LIN {X 0,Y 509.826,Z 394.48,A -85,B 0,C 180,E1 -5633.741,E2 -5633.741} C_VEL
LIN {X 0,Y 509.161,Z 394.559,A -85,B 0,C 180,E1 -5634.401,E2 -5634.401} C_VEL
LIN {X 0,Y 506.342,Z 394.916,A -85,B 0,C 180,E1 -5635.473,E2 -5635.473} C_VEL
LIN {X 0,Y 503.949,Z 395.212,A -85,B 0,C 180,E1 -5636.336,E2 -5636.336} C_VEL
LIN {X 0,Y 502.9,Z 395.339,A -85,B 0,C 180,E1 -5637.003,E2 -5637.003} C_VEL
LIN {X 0,Y 502.803,Z 395.349,A -85,B 0,C 180,E1 -5637.228,E2 -5637.228} C_VEL
LIN {X 0,Y 502.809,Z 395.349,A -85,B 0,C 180,E1 -5640.065,E2 -5640.065} C_VEL
LIN {X 0,Y 502.83,Z 395.345,A -85,B 0,C 180,E1 -5642.534,E2 -5642.534} C_VEL
LIN {X 0,Y 502.824,Z 395.354,A -85,B 0,C 180,E1 -5645.299,E2 -5645.299} C_VEL
LIN {X 0,Y 502.789,Z 395.353,A -85,B 0,C 180,E1 -5647.827,E2 -5647.827} C_VEL
LIN {X 0,Y 502.82,Z 395.346,A -85,B 0,C 180,E1 -5650.4,E2 -5650.4} C_VEL
LIN {X 0,Y 502.83,Z 395.351,A -85,B 0,C 180,E1 -5652.932,E2 -5652.932} C_VEL
LIN {X 0,Y 502.841,Z 395.351,A -85,B 0,C 180,E1 -5655.429,E2 -5655.429} C_VEL
LIN {X 0,Y 502.874,Z 395.344,A -85,B 0,C 180,E1 -5658.717,E2 -5658.717} C_VEL
LIN {X 0,Y 502.898,Z 395.34,A -85,B 0,C 180,E1 -5661.967,E2 -5661.967} C_VEL
LIN {X 0,Y 502.939,Z 395.335,A -85,B 0,C 180,E1 -5664.387,E2 -5664.387} C_VEL
LIN {X 0,Y 503.023,Z 395.325,A -85,B 0,C 180,E1 -5667.598,E2 -5667.598} C_VEL
LIN {X 0,Y 503.025,Z 395.324,A -85,B 0,C 180,E1 -5670,E2 -5670} C_VEL
LIN {X 0,Y 503.023,Z 395.325,A -85,B 0,C 180,E1 -5672.402,E2 -5672.402} C_VEL
LIN {X 0,Y 502.939,Z 395.335,A -85,B 0,C 180,E1 -5675.614,E2 -5675.614} C_VEL
LIN {X 0,Y 502.899,Z 395.339,A -85,B 0,C 180,E1 -5678.033,E2 -5678.033} C_VEL
LIN {X 0,Y 502.875,Z 395.344,A -85,B 0,C 180,E1 -5681.283,E2 -5681.283} C_VEL
LIN {X 0,Y 502.841,Z 395.351,A -85,B 0,C 180,E1 -5684.571,E2 -5684.571} C_VEL
LIN {X 0,Y 502.858,Z 395.344,A -85,B 0,C 180,E1 -5687.907,E2 -5687.907} C_VEL
LIN {X 0,Y 502.825,Z 395.353,A -85,B 0,C 180,E1 -5690.536,E2 -5690.536} C_VEL
LIN {X 0,Y 502.793,Z 395.353,A -85,B 0,C 180,E1 -5693.04,E2 -5693.04} C_VEL
LIN {X 0,Y 502.838,Z 395.344,A -85,B 0,C 180,E1 -5695.675,E2 -5695.675} C_VEL
LIN {X 0,Y 502.837,Z 395.35,A -85,B 0,C 180,E1 -5698.373,E2 -5698.373} C_VEL
LIN {X 0,Y 502.792,Z 395.35,A -85,B 0,C 180,E1 -5701.5,E2 -5701.5} C_VEL
LIN {X 0,Y 502.802,Z 395.358,A -85,B 0,C 180,E1 -5704.445,E2 -5704.445} C_VEL
LIN {X 0,Y 502.777,Z 395.352,A -85,B 0,C 180,E1 -5707.179,E2 -5707.179} C_VEL
LIN {X 0,Y 502.817,Z 395.35,A -85,B 0,C 180,E1 -5710.012,E2 -5710.012} C_VEL
LIN {X 0,Y 502.819,Z 395.353,A -85,B 0,C 180,E1 -5712.202,E2 -5712.202} C_VEL
LIN {X 0,Y 502.795,Z 395.35,A -85,B 0,C 180,E1 -5715.468,E2 -5715.468} C_VEL
LIN {X 0,Y 502.815,Z 395.348,A -85,B 0,C 180,E1 -5718.934,E2 -5718.934} C_VEL
LIN {X 0,Y 502.789,Z 395.357,A -85,B 0,C 180,E1 -5722.046,E2 -5722.046} C_VEL
LIN {X 0,Y 502.804,Z 395.349,A -85,B 0,C 180,E1 -5725.035,E2 -5725.035} C_VEL
LIN {X 0,Y 502.783,Z 395.357,A -85,B 0,C 180,E1 -5727.916,E2 -5727.916} C_VEL
LIN {X 0,Y 502.834,Z 395.346,A -85,B 0,C 180,E1 -5730.713,E2 -5730.713} C_VEL
LIN {X 0,Y 502.857,Z 395.343,A -85,B 0,C 180,E1 -5733.439,E2 -5733.439} C_VEL
LIN {X 0,Y 502.787,Z 395.358,A -85,B 0,C 180,E1 -5736.087,E2 -5736.087} C_VEL
LIN {X 0,Y 502.778,Z 395.352,A -85,B 0,C 180,E1 -5738.689,E2 -5738.689} C_VEL
LIN {X 0,Y 502.826,Z 395.347,A -85,B 0,C 180,E1 -5741.249,E2 -5741.249} C_VEL
LIN {X 0,Y 502.819,Z 395.354,A -85,B 0,C 180,E1 -5743.768,E2 -5743.768} C_VEL
LIN {X 0,Y 502.827,Z 395.349,A -85,B 0,C 180,E1 -5746.255,E2 -5746.255} C_VEL
LIN {X 0,Y 502.872,Z 395.34,A -85,B 0,C 180,E1 -5748.717,E2 -5748.717} C_VEL
LIN {X 0,Y 502.897,Z 395.342,A -85,B 0,C 180,E1 -5751.967,E2 -5751.967} C_VEL
LIN {X 0,Y 502.934,Z 395.333,A -85,B 0,C 180,E1 -5754.387,E2 -5754.387} C_VEL
LIN {X 0,Y 503.021,Z 395.33,A -85,B 0,C 180,E1 -5757.598,E2 -5757.598} C_VEL
LIN {X 0,Y 503.023,Z 395.325,A -85,B 0,C 180,E1 -5760,E2 -5760} C_VEL
LIN {X 0,Y 503.021,Z 395.322,A -85,B 0,C 180,E1 -5762.403,E2 -5762.403} C_VEL
LIN {X 0,Y 502.935,Z 395.34,A -85,B 0,C 180,E1 -5765.614,E2 -5765.614} C_VEL
LIN {X 0,Y 502.898,Z 395.339,A -85,B 0,C 180,E1 -5768.034,E2 -5768.034} C_VEL
LIN {X 0,Y 502.874,Z 395.346,A -85,B 0,C 180,E1 -5771.284,E2 -5771.284} C_VEL
LIN {X 0,Y 502.842,Z 395.344,A -85,B 0,C 180,E1 -5774.571,E2 -5774.571} C_VEL
LIN {X 0,Y 502.859,Z 395.343,A -85,B 0,C 180,E1 -5777.907,E2 -5777.907} C_VEL
LIN {X 0,Y 502.826,Z 395.346,A -85,B 0,C 180,E1 -5780.537,E2 -5780.537} C_VEL
LIN {X 0,Y 502.792,Z 395.356,A -85,B 0,C 180,E1 -5783.041,E2 -5783.041} C_VEL
LIN {X 0,Y 502.838,Z 395.347,A -85,B 0,C 180,E1 -5785.676,E2 -5785.676} C_VEL
LIN {X 0,Y 502.839,Z 395.345,A -85,B 0,C 180,E1 -5788.373,E2 -5788.373} C_VEL
LIN {X 0,Y 502.795,Z 395.353,A -85,B 0,C 180,E1 -5791.5,E2 -5791.5} C_VEL
LIN {X 0,Y 502.805,Z 395.35,A -85,B 0,C 180,E1 -5794.445,E2 -5794.445} C_VEL
LIN {X 0,Y 502.781,Z 395.36,A -85,B 0,C 180,E1 -5797.179,E2 -5797.179} C_VEL
LIN {X 0,Y 502.788,Z 395.355,A -85,B 0,C 180,E1 -5800.016,E2 -5800.016} C_VEL
LIN {X 0,Y 502.802,Z 395.354,A -85,B 0,C 180,E1 -5802.2,E2 -5802.2} C_VEL
LIN {X 0,Y 502.772,Z 395.36,A -85,B 0,C 180,E1 -5803.375,E2 -5803.375} C_VEL
LIN {X 0,Y 502.912,Z 396.072,A -85,B 0,C 180,E1 -5804.545,E2 -5804.545} C_VEL
LIN {X 0,Y 503.525,Z 400.319,A -85,B 0,C 180,E1 -5807.711,E2 -5807.711} C_VEL
LIN {X 0,Y 503.571,Z 403.923,A -85,B 0,C 180,E1 -5810.139,E2 -5810.139} C_VEL
LIN {X 0,Y 503.281,Z 408.665,A -85,B 0,C 180,E1 -5813.097,E2 -5813.097} C_VEL
LIN {X 0,Y 503.066,Z 413.701,A -85,B 0,C 180,E1 -5816.027,E2 -5816.027} C_VEL
LIN {X 0,Y 502.877,Z 418.836,A -85,B 0,C 180,E1 -5818.863,E2 -5818.863} C_VEL
LIN {X 0,Y 502.696,Z 424.321,A -85,B 0,C 180,E1 -5821.737,E2 -5821.737} C_VEL
LIN {X 0,Y 502.579,Z 429.398,A -85,B 0,C 180,E1 -5824.31,E2 -5824.31} C_VEL
LIN {X 0,Y 502.486,Z 435.794,A -85,B 0,C 180,E1 -5827.385,E2 -5827.385} C_VEL
LIN {X 0,Y 502.376,Z 442.071,A -85,B 0,C 180,E1 -5830.382,E2 -5830.382} C_VEL
LIN {X 0,Y 502.245,Z 447.46,A -85,B 0,C 180,E1 -5832.911,E2 -5832.911} C_VEL
LIN {X 0,Y 502.241,Z 453.523,A -85,B 0,C 180,E1 -5835.722,E2 -5835.722} C_VEL
LIN {X 0,Y 504.317,Z 465.721,A -85,B 0,C 180,E1 -5836.09,E2 -5836.09} C_VEL
LIN {X 0,Y 504.61,Z 469.05,A -85,B 0,C 180,E1 -5836.201,E2 -5836.201} C_VEL
LIN {X 0,Y 504.336,Z 481.375,A -85,B 0,C 180,E1 -5836.707,E2 -5836.707} C_VEL
LIN {X 0,Y 504.044,Z 491.745,A -85,B 0,C 180,E1 -5837.267,E2 -5837.267} C_VEL
LIN {X 0,Y 503.765,Z 501.474,A -85,B 0,C 180,E1 -5837.921,E2 -5837.921} C_VEL
LIN {X 0,Y 503.465,Z 510.173,A -85,B 0,C 180,E1 -5838.628,E2 -5838.628} C_VEL
LIN {X 0,Y 503.19,Z 517.54,A -85,B 0,C 180,E1 -5839.335,E2 -5839.335} C_VEL
LIN {X 0,Y 502.948,Z 524.728,A -85,B 0,C 180,E1 -5840.144,E2 -5840.144} C_VEL
LIN {X 0,Y 502.683,Z 532.274,A -85,B 0,C 180,E1 -5841.153,E2 -5841.153} C_VEL
LIN {X 0,Y 502.471,Z 538.564,A -85,B 0,C 180,E1 -5842.162,E2 -5842.162} C_VEL
LIN {X 0,Y 502.317,Z 543.988,A -85,B 0,C 180,E1 -5843.21,E2 -5843.21} C_VEL
LIN {X 0,Y 502.256,Z 548.894,A -85,B 0,C 180,E1 -5844.379,E2 -5844.379} C_VEL
LIN {X 0,Y 502.128,Z 552.85,A -85,B 0,C 180,E1 -5845.585,E2 -5845.585} C_VEL
LIN {X 0,Y 502.121,Z 555.772,A -85,B 0,C 180,E1 -5846.79,E2 -5846.79} C_VEL
LIN {X 0,Y 502.036,Z 558.196,A -85,B 0,C 180,E1 -5848.395,E2 -5848.395} C_VEL
LIN {X 0,Y 501.991,Z 558.78,A -85,B 0,C 180,E1 -5849.198,E2 -5849.198} C_VEL
LIN {X 0,Y 501.991,Z 558.78,A -85,B 0,C 180,E1 -5850.802,E2 -5850.802} C_VEL
LIN {X 0,Y 502.036,Z 558.196,A -85,B 0,C 180,E1 -5851.604,E2 -5851.604} C_VEL
LIN {X 0,Y 502.121,Z 555.772,A -85,B 0,C 180,E1 -5853.209,E2 -5853.209} C_VEL
LIN {X 0,Y 502.128,Z 552.851,A -85,B 0,C 180,E1 -5854.415,E2 -5854.415} C_VEL
LIN {X 0,Y 502.256,Z 548.896,A -85,B 0,C 180,E1 -5855.621,E2 -5855.621} C_VEL
LIN {X 0,Y 502.317,Z 543.989,A -85,B 0,C 180,E1 -5856.789,E2 -5856.789} C_VEL
LIN {X 0,Y 502.47,Z 538.566,A -85,B 0,C 180,E1 -5857.838,E2 -5857.838} C_VEL
LIN {X 0,Y 502.682,Z 532.277,A -85,B 0,C 180,E1 -5858.846,E2 -5858.846} C_VEL
LIN {X 0,Y 502.947,Z 524.731,A -85,B 0,C 180,E1 -5859.856,E2 -5859.856} C_VEL
LIN {X 0,Y 503.219,Z 515.622,A -85,B 0,C 180,E1 -5860.867,E2 -5860.867} C_VEL
LIN {X 0,Y 503.674,Z 504.176,A -85,B 0,C 180,E1 -5861.877,E2 -5861.877} C_VEL
LIN {X 0,Y 503.936,Z 494.382,A -85,B 0,C 180,E1 -5862.57,E2 -5862.57} C_VEL
LIN {X 0,Y 504.202,Z 484.399,A -85,B 0,C 180,E1 -5863.142,E2 -5863.142} C_VEL
LIN {X 0,Y 504.491,Z 474.335,A -85,B 0,C 180,E1 -5863.596,E2 -5863.596} C_VEL
LIN {X 0,Y 504.472,Z 466.607,A -85,B 0,C 180,E1 -5863.879,E2 -5863.879} C_VEL
LIN {X 0,Y 502.563,Z 455.442,A -85,B 0,C 180,E1 -5864.226,E2 -5864.226} C_VEL
LIN {X 0,Y 502.244,Z 453.524,A -85,B 0,C 180,E1 -5864.278,E2 -5864.278} C_VEL
LIN {X 0,Y 502.244,Z 447.461,A -85,B 0,C 180,E1 -5867.089,E2 -5867.089} C_VEL
LIN {X 0,Y 502.43,Z 440.391,A -85,B 0,C 180,E1 -5870.413,E2 -5870.413} C_VEL
LIN {X 0,Y 502.482,Z 434.885,A -85,B 0,C 180,E1 -5873.055,E2 -5873.055} C_VEL
LIN {X 0,Y 502.578,Z 429.398,A -85,B 0,C 180,E1 -5875.689,E2 -5875.689} C_VEL
LIN {X 0,Y 502.701,Z 424.094,A -85,B 0,C 180,E1 -5878.381,E2 -5878.381} C_VEL
LIN {X 0,Y 502.875,Z 418.832,A -85,B 0,C 180,E1 -5881.137,E2 -5881.137} C_VEL
LIN {X 0,Y 503.064,Z 413.669,A -85,B 0,C 180,E1 -5883.973,E2 -5883.973} C_VEL
LIN {X 0,Y 503.328,Z 408.065,A -85,B 0,C 180,E1 -5887.26,E2 -5887.26} C_VEL
LIN {X 0,Y 503.544,Z 403.787,A -85,B 0,C 180,E1 -5889.942,E2 -5889.942} C_VEL
LIN {X 0,Y 503.522,Z 400.313,A -85,B 0,C 180,E1 -5892.289,E2 -5892.289} C_VEL
LIN {X 0,Y 502.909,Z 396.09,A -85,B 0,C 180,E1 -5895.455,E2 -5895.455} C_VEL
LIN {X 0,Y 502.771,Z 395.359,A -85,B 0,C 180,E1 -5896.768,E2 -5896.768} C_VEL
LIN {X 0,Y 502.817,Z 395.356,A -85,B 0,C 180,E1 -5899.004,E2 -5899.004} C_VEL
LIN {X 0,Y 502.791,Z 395.353,A -85,B 0,C 180,E1 -5902.045,E2 -5902.045} C_VEL
LIN {X 0,Y 502.806,Z 395.357,A -85,B 0,C 180,E1 -5905.034,E2 -5905.034} C_VEL
LIN {X 0,Y 502.784,Z 395.351,A -85,B 0,C 180,E1 -5907.915,E2 -5907.915} C_VEL
LIN {X 0,Y 502.835,Z 395.352,A -85,B 0,C 180,E1 -5910.712,E2 -5910.712} C_VEL
LIN {X 0,Y 502.858,Z 395.343,A -85,B 0,C 180,E1 -5913.438,E2 -5913.438} C_VEL
LIN {X 0,Y 502.787,Z 395.352,A -85,B 0,C 180,E1 -5916.086,E2 -5916.086} C_VEL
LIN {X 0,Y 502.778,Z 395.36,A -85,B 0,C 180,E1 -5918.688,E2 -5918.688} C_VEL
LIN {X 0,Y 502.826,Z 395.347,A -85,B 0,C 180,E1 -5921.248,E2 -5921.248} C_VEL
LIN {X 0,Y 502.818,Z 395.347,A -85,B 0,C 180,E1 -5923.767,E2 -5923.767} C_VEL
LIN {X 0,Y 502.826,Z 395.35,A -85,B 0,C 180,E1 -5926.254,E2 -5926.254} C_VEL
LIN {X 0,Y 502.871,Z 395.347,A -85,B 0,C 180,E1 -5928.716,E2 -5928.716} C_VEL
LIN {X 0,Y 502.896,Z 395.339,A -85,B 0,C 180,E1 -5931.966,E2 -5931.966} C_VEL
LIN {X 0,Y 502.933,Z 395.34,A -85,B 0,C 180,E1 -5934.386,E2 -5934.386} C_VEL
LIN {X 0,Y 503.019,Z 395.322,A -85,B 0,C 180,E1 -5937.597,E2 -5937.597} C_VEL
LIN {X 0,Y 503.02,Z 395.325,A -85,B 0,C 180,E1 -5940,E2 -5940} C_VEL
LIN {X 0,Y 503.019,Z 395.33,A -85,B 0,C 180,E1 -5942.402,E2 -5942.402} C_VEL
LIN {X 0,Y 502.933,Z 395.333,A -85,B 0,C 180,E1 -5945.613,E2 -5945.613} C_VEL
LIN {X 0,Y 502.895,Z 395.343,A -85,B 0,C 180,E1 -5948.033,E2 -5948.033} C_VEL
LIN {X 0,Y 502.87,Z 395.34,A -85,B 0,C 180,E1 -5951.283,E2 -5951.283} C_VEL
LIN {X 0,Y 502.838,Z 395.347,A -85,B 0,C 180,E1 -5954.571,E2 -5954.571} C_VEL
LIN {X 0,Y 502.854,Z 395.348,A -85,B 0,C 180,E1 -5957.907,E2 -5957.907} C_VEL
LIN {X 0,Y 502.82,Z 395.349,A -85,B 0,C 180,E1 -5960.536,E2 -5960.536} C_VEL
LIN {X 0,Y 502.789,Z 395.35,A -85,B 0,C 180,E1 -5963.04,E2 -5963.04} C_VEL
LIN {X 0,Y 502.834,Z 395.349,A -85,B 0,C 180,E1 -5965.675,E2 -5965.675} C_VEL
LIN {X 0,Y 502.835,Z 395.348,A -85,B 0,C 180,E1 -5968.372,E2 -5968.372} C_VEL
LIN {X 0,Y 502.79,Z 395.354,A -85,B 0,C 180,E1 -5971.5,E2 -5971.5} C_VEL
LIN {X 0,Y 502.8,Z 395.351,A -85,B 0,C 180,E1 -5974.445,E2 -5974.445} C_VEL
LIN {X 0,Y 502.774,Z 395.353,A -85,B 0,C 180,E1 -5977.178,E2 -5977.178} C_VEL
LIN {X 0,Y 502.819,Z 395.352,A -85,B 0,C 180,E1 -5980.012,E2 -5980.012} C_VEL
LIN {X 0,Y 502.822,Z 395.349,A -85,B 0,C 180,E1 -5982.203,E2 -5982.203} C_VEL
LIN {X 0,Y 502.794,Z 395.355,A -85,B 0,C 180,E1 -5985.468,E2 -5985.468} C_VEL
LIN {X 0,Y 502.829,Z 395.351,A -85,B 0,C 180,E1 -5987.865,E2 -5987.865} C_VEL
LIN {X 0,Y 502.803,Z 395.35,A -85,B 0,C 180,E1 -5991.025,E2 -5991.025} C_VEL
LIN {X 0,Y 502.78,Z 395.353,A -85,B 0,C 180,E1 -5994.167,E2 -5994.167} C_VEL
LIN {X 0,Y 502.803,Z 395.349,A -85,B 0,C 180,E1 -5997.228,E2 -5997.228} C_VEL
LIN {X 0,Y 502.104,Z 395.439,A -85,B 0,C 180,E1 -5997.897,E2 -5997.897} C_VEL
LIN {X 0,Y 499.238,Z 395.795,A -85,B 0,C 180,E1 -5998.983,E2 -5998.983} C_VEL
LIN {X 0,Y 496.842,Z 396.095,A -85,B 0,C 180,E1 -5999.858,E2 -5999.858} C_VEL
LIN {X 0,Y 495.826,Z 396.218,A -85,B 0,C 180,E1 -6000.533,E2 -6000.533} C_VEL
LIN {X 0,Y 495.748,Z 396.228,A -85,B 0,C 180,E1 -6000.762,E2 -6000.762} C_VEL
LIN {X 0,Y 495.794,Z 396.224,A -85,B 0,C 180,E1 -6003.933,E2 -6003.933} C_VEL
LIN {X 0,Y 495.753,Z 396.232,A -85,B 0,C 180,E1 -6007.14,E2 -6007.14} C_VEL
LIN {X 0,Y 495.773,Z 396.225,A -85,B 0,C 180,E1 -6010.11,E2 -6010.11} C_VEL
LIN {X 0,Y 495.782,Z 396.227,A -85,B 0,C 180,E1 -6012.682,E2 -6012.682} C_VEL
LIN {X 0,Y 495.786,Z 396.232,A -85,B 0,C 180,E1 -6015.217,E2 -6015.217} C_VEL
LIN {X 0,Y 495.848,Z 396.218,A -85,B 0,C 180,E1 -6018.555,E2 -6018.555} C_VEL
LIN {X 0,Y 495.87,Z 396.216,A -85,B 0,C 180,E1 -6021.852,E2 -6021.852} C_VEL
LIN {X 0,Y 495.896,Z 396.212,A -85,B 0,C 180,E1 -6024.307,E2 -6024.307} C_VEL
LIN {X 0,Y 495.991,Z 396.202,A -85,B 0,C 180,E1 -6027.564,E2 -6027.564} C_VEL
LIN {X 0,Y 495.996,Z 396.2,A -85,B 0,C 180,E1 -6030,E2 -6030} C_VEL
LIN {X 0,Y 495.992,Z 396.202,A -85,B 0,C 180,E1 -6032.436,E2 -6032.436} C_VEL
LIN {X 0,Y 495.897,Z 396.212,A -85,B 0,C 180,E1 -6035.694,E2 -6035.694} C_VEL
LIN {X 0,Y 495.87,Z 396.216,A -85,B 0,C 180,E1 -6038.148,E2 -6038.148} C_VEL
LIN {X 0,Y 495.849,Z 396.218,A -85,B 0,C 180,E1 -6041.445,E2 -6041.445} C_VEL
LIN {X 0,Y 495.787,Z 396.232,A -85,B 0,C 180,E1 -6044.783,E2 -6044.783} C_VEL
LIN {X 0,Y 495.783,Z 396.227,A -85,B 0,C 180,E1 -6047.319,E2 -6047.319} C_VEL
LIN {X 0,Y 495.774,Z 396.225,A -85,B 0,C 180,E1 -6049.89,E2 -6049.89} C_VEL
LIN {X 0,Y 495.754,Z 396.232,A -85,B 0,C 180,E1 -6052.86,E2 -6052.86} C_VEL
LIN {X 0,Y 495.796,Z 396.224,A -85,B 0,C 180,E1 -6056.067,E2 -6056.067} C_VEL
LIN {X 0,Y 495.769,Z 396.23,A -85,B 0,C 180,E1 -6058.815,E2 -6058.815} C_VEL
LIN {X 0,Y 495.754,Z 396.227,A -85,B 0,C 180,E1 -6061.726,E2 -6061.726} C_VEL
LIN {X 0,Y 495.772,Z 396.23,A -85,B 0,C 180,E1 -6064.695,E2 -6064.695} C_VEL
LIN {X 0,Y 495.727,Z 396.23,A -85,B 0,C 180,E1 -6067.561,E2 -6067.561} C_VEL
LIN {X 0,Y 495.775,Z 396.228,A -85,B 0,C 180,E1 -6070.699,E2 -6070.699} C_VEL
LIN {X 0,Y 495.73,Z 396.231,A -85,B 0,C 180,E1 -6073.696,E2 -6073.696} C_VEL
LIN {X 0,Y 495.723,Z 396.239,A -85,B 0,C 180,E1 -6076.305,E2 -6076.305} C_VEL
LIN {X 0,Y 495.762,Z 396.226,A -85,B 0,C 180,E1 -6079.3,E2 -6079.3} C_VEL
LIN {X 0,Y 495.727,Z 396.235,A -85,B 0,C 180,E1 -6082.439,E2 -6082.439} C_VEL
LIN {X 0,Y 495.78,Z 396.224,A -85,B 0,C 180,E1 -6085.458,E2 -6085.458} C_VEL
LIN {X 0,Y 495.755,Z 396.232,A -85,B 0,C 180,E1 -6088.364,E2 -6088.364} C_VEL
LIN {X 0,Y 495.785,Z 396.225,A -85,B 0,C 180,E1 -6091.506,E2 -6091.506} C_VEL
LIN {X 0,Y 495.786,Z 396.23,A -85,B 0,C 180,E1 -6093.932,E2 -6093.932} C_VEL
LIN {X 0,Y 495.76,Z 396.226,A -85,B 0,C 180,E1 -6097.138,E2 -6097.138} C_VEL
LIN {X 0,Y 495.767,Z 396.231,A -85,B 0,C 180,E1 -6100.11,E2 -6100.11} C_VEL
LIN {X 0,Y 495.783,Z 396.223,A -85,B 0,C 180,E1 -6102.682,E2 -6102.682} C_VEL
LIN {X 0,Y 495.785,Z 396.224,A -85,B 0,C 180,E1 -6105.218,E2 -6105.218} C_VEL
LIN {X 0,Y 495.847,Z 396.216,A -85,B 0,C 180,E1 -6108.555,E2 -6108.555} C_VEL
LIN {X 0,Y 495.869,Z 396.22,A -85,B 0,C 180,E1 -6111.852,E2 -6111.852} C_VEL
LIN {X 0,Y 495.892,Z 396.211,A -85,B 0,C 180,E1 -6114.307,E2 -6114.307} C_VEL
LIN {X 0,Y 495.989,Z 396.205,A -85,B 0,C 180,E1 -6117.564,E2 -6117.564} C_VEL
LIN {X 0,Y 495.994,Z 396.2,A -85,B 0,C 180,E1 -6120,E2 -6120} C_VEL
LIN {X 0,Y 495.99,Z 396.198,A -85,B 0,C 180,E1 -6122.437,E2 -6122.437} C_VEL
LIN {X 0,Y 495.893,Z 396.216,A -85,B 0,C 180,E1 -6125.694,E2 -6125.694} C_VEL
LIN {X 0,Y 495.87,Z 396.213,A -85,B 0,C 180,E1 -6128.148,E2 -6128.148} C_VEL
LIN {X 0,Y 495.848,Z 396.224,A -85,B 0,C 180,E1 -6131.446,E2 -6131.446} C_VEL
LIN {X 0,Y 495.787,Z 396.224,A -85,B 0,C 180,E1 -6134.783,E2 -6134.783} C_VEL
LIN {X 0,Y 495.785,Z 396.232,A -85,B 0,C 180,E1 -6137.319,E2 -6137.319} C_VEL
LIN {X 0,Y 495.769,Z 396.226,A -85,B 0,C 180,E1 -6139.891,E2 -6139.891} C_VEL
LIN {X 0,Y 495.759,Z 396.229,A -85,B 0,C 180,E1 -6142.862,E2 -6142.862} C_VEL
LIN {X 0,Y 495.789,Z 396.223,A -85,B 0,C 180,E1 -6146.068,E2 -6146.068} C_VEL
LIN {X 0,Y 495.77,Z 396.229,A -85,B 0,C 180,E1 -6148.815,E2 -6148.815} C_VEL
LIN {X 0,Y 495.757,Z 396.228,A -85,B 0,C 180,E1 -6151.727,E2 -6151.727} C_VEL
LIN {X 0,Y 495.775,Z 396.228,A -85,B 0,C 180,E1 -6154.696,E2 -6154.696} C_VEL
LIN {X 0,Y 495.731,Z 396.235,A -85,B 0,C 180,E1 -6157.562,E2 -6157.562} C_VEL
LIN {X 0,Y 495.767,Z 396.233,A -85,B 0,C 180,E1 -6160.7,E2 -6160.7} C_VEL
LIN {X 0,Y 495.748,Z 396.299,A -85,B 0,C 180,E1 -6163.698,E2 -6163.698} C_VEL
LIN {X 0,Y 496.26,Z 399.542,A -85,B 0,C 180,E1 -6166.242,E2 -6166.242} C_VEL
LIN {X 0,Y 496.607,Z 402.78,A -85,B 0,C 180,E1 -6168.596,E2 -6168.596} C_VEL
LIN {X 0,Y 496.465,Z 407.14,A -85,B 0,C 180,E1 -6171.475,E2 -6171.475} C_VEL
LIN {X 0,Y 496.125,Z 412.071,A -85,B 0,C 180,E1 -6174.494,E2 -6174.494} C_VEL
LIN {X 0,Y 495.938,Z 417.147,A -85,B 0,C 180,E1 -6177.419,E2 -6177.419} C_VEL
LIN {X 0,Y 495.752,Z 422.337,A -85,B 0,C 180,E1 -6180.253,E2 -6180.253} C_VEL
LIN {X 0,Y 495.609,Z 428.151,A -85,B 0,C 180,E1 -6183.301,E2 -6183.301} C_VEL
LIN {X 0,Y 495.465,Z 432.972,A -85,B 0,C 180,E1 -6185.71,E2 -6185.71} C_VEL
LIN {X 0,Y 495.402,Z 438.478,A -85,B 0,C 180,E1 -6188.356,E2 -6188.356} C_VEL
LIN {X 0,Y 495.277,Z 443.867,A -85,B 0,C 180,E1 -6190.951,E2 -6190.951} C_VEL
LIN {X 0,Y 495.143,Z 449.257,A -85,B 0,C 180,E1 -6193.508,E2 -6193.508} C_VEL
LIN {X 0,Y 495.174,Z 453.523,A -85,B 0,C 180,E1 -6195.514,E2 -6195.514} C_VEL
LIN {X 0,Y 497.243,Z 465.704,A -85,B 0,C 180,E1 -6195.889,E2 -6195.889} C_VEL
LIN {X 0,Y 497.737,Z 469.054,A -85,B 0,C 180,E1 -6196.007,E2 -6196.007} C_VEL
LIN {X 0,Y 497.444,Z 481.366,A -85,B 0,C 180,E1 -6196.519,E2 -6196.519} C_VEL
LIN {X 0,Y 497.093,Z 491.986,A -85,B 0,C 180,E1 -6197.101,E2 -6197.101} C_VEL
LIN {X 0,Y 496.807,Z 501.467,A -85,B 0,C 180,E1 -6197.749,E2 -6197.749} C_VEL
LIN {X 0,Y 496.491,Z 510.167,A -85,B 0,C 180,E1 -6198.466,E2 -6198.466} C_VEL
LIN {X 0,Y 496.186,Z 517.535,A -85,B 0,C 180,E1 -6199.183,E2 -6199.183} C_VEL
LIN {X 0,Y 495.929,Z 524.724,A -85,B 0,C 180,E1 -6200.003,E2 -6200.003} C_VEL
LIN {X 0,Y 495.634,Z 532.27,A -85,B 0,C 180,E1 -6201.026,E2 -6201.026} C_VEL
LIN {X 0,Y 495.404,Z 538.559,A -85,B 0,C 180,E1 -6202.049,E2 -6202.049} C_VEL
LIN {X 0,Y 495.248,Z 543.983,A -85,B 0,C 180,E1 -6203.113,E2 -6203.113} C_VEL
LIN {X 0,Y 495.174,Z 548.89,A -85,B 0,C 180,E1 -6204.298,E2 -6204.298} C_VEL
LIN {X 0,Y 495.029,Z 552.846,A -85,B 0,C 180,E1 -6205.521,E2 -6205.521} C_VEL
LIN {X 0,Y 495.043,Z 555.769,A -85,B 0,C 180,E1 -6206.744,E2 -6206.744} C_VEL
LIN {X 0,Y 494.961,Z 558.195,A -85,B 0,C 180,E1 -6208.373,E2 -6208.373} C_VEL
LIN {X 0,Y 494.911,Z 558.779,A -85,B 0,C 180,E1 -6209.186,E2 -6209.186} C_VEL
LIN {X 0,Y 494.911,Z 558.78,A -85,B 0,C 180,E1 -6210.813,E2 -6210.813} C_VEL
LIN {X 0,Y 494.961,Z 558.195,A -85,B 0,C 180,E1 -6211.627,E2 -6211.627} C_VEL
LIN {X 0,Y 495.043,Z 555.77,A -85,B 0,C 180,E1 -6213.255,E2 -6213.255} C_VEL
LIN {X 0,Y 495.028,Z 552.847,A -85,B 0,C 180,E1 -6214.478,E2 -6214.478} C_VEL
LIN {X 0,Y 495.175,Z 548.891,A -85,B 0,C 180,E1 -6215.702,E2 -6215.702} C_VEL
LIN {X 0,Y 495.247,Z 543.985,A -85,B 0,C 180,E1 -6216.887,E2 -6216.887} C_VEL
LIN {X 0,Y 495.403,Z 538.561,A -85,B 0,C 180,E1 -6217.95,E2 -6217.95} C_VEL
LIN {X 0,Y 495.634,Z 532.272,A -85,B 0,C 180,E1 -6218.973,E2 -6218.973} C_VEL
LIN {X 0,Y 495.929,Z 524.727,A -85,B 0,C 180,E1 -6219.997,E2 -6219.997} C_VEL
LIN {X 0,Y 496.243,Z 515.62,A -85,B 0,C 180,E1 -6221.022,E2 -6221.022} C_VEL
LIN {X 0,Y 496.723,Z 504.168,A -85,B 0,C 180,E1 -6222.045,E2 -6222.045} C_VEL
LIN {X 0,Y 496.982,Z 494.866,A -85,B 0,C 180,E1 -6222.718,E2 -6222.718} C_VEL
LIN {X 0,Y 497.274,Z 484.389,A -85,B 0,C 180,E1 -6223.329,E2 -6223.329} C_VEL
LIN {X 0,Y 497.606,Z 474.326,A -85,B 0,C 180,E1 -6223.788,E2 -6223.788} C_VEL
LIN {X 0,Y 497.545,Z 467.464,A -85,B 0,C 180,E1 -6224.05,E2 -6224.05} C_VEL
LIN {X 0,Y 495.519,Z 455.49,A -85,B 0,C 180,E1 -6224.431,E2 -6224.431} C_VEL
LIN {X 0,Y 495.167,Z 453.524,A -85,B 0,C 180,E1 -6224.486,E2 -6224.486} C_VEL
LIN {X 0,Y 495.217,Z 445.99,A -85,B 0,C 180,E1 -6228.038,E2 -6228.038} C_VEL
LIN {X 0,Y 495.377,Z 440.275,A -85,B 0,C 180,E1 -6230.773,E2 -6230.773} C_VEL
LIN {X 0,Y 495.43,Z 434.813,A -85,B 0,C 180,E1 -6233.403,E2 -6233.403} C_VEL
LIN {X 0,Y 495.538,Z 429.353,A -85,B 0,C 180,E1 -6236.082,E2 -6236.082} C_VEL
LIN {X 0,Y 495.675,Z 424.091,A -85,B 0,C 180,E1 -6238.82,E2 -6238.82} C_VEL
LIN {X 0,Y 495.868,Z 418.623,A -85,B 0,C 180,E1 -6241.746,E2 -6241.746} C_VEL
LIN {X 0,Y 496.077,Z 413.358,A -85,B 0,C 180,E1 -6244.745,E2 -6244.745} C_VEL
LIN {X 0,Y 496.33,Z 408.7,A -85,B 0,C 180,E1 -6247.537,E2 -6247.537} C_VEL
LIN {X 0,Y 496.534,Z 404.625,A -85,B 0,C 180,E1 -6250.153,E2 -6250.153} C_VEL
LIN {X 0,Y 496.584,Z 402.356,A -85,B 0,C 180,E1 -6251.695,E2 -6251.695} C_VEL
LIN {X 0,Y 496.224,Z 399.276,A -85,B 0,C 180,E1 -6253.945,E2 -6253.945} C_VEL
LIN {X 0,Y 495.746,Z 396.296,A -85,B 0,C 180,E1 -6256.302,E2 -6256.302} C_VEL
LIN {X 0,Y 495.764,Z 396.233,A -85,B 0,C 180,E1 -6259.299,E2 -6259.299} C_VEL
LIN {X 0,Y 495.729,Z 396.235,A -85,B 0,C 180,E1 -6262.438,E2 -6262.438} C_VEL
LIN {X 0,Y 495.782,Z 396.226,A -85,B 0,C 180,E1 -6265.457,E2 -6265.457} C_VEL
LIN {X 0,Y 495.756,Z 396.229,A -85,B 0,C 180,E1 -6268.363,E2 -6268.363} C_VEL
LIN {X 0,Y 495.786,Z 396.224,A -85,B 0,C 180,E1 -6271.505,E2 -6271.505} C_VEL
LIN {X 0,Y 495.786,Z 396.223,A -85,B 0,C 180,E1 -6273.931,E2 -6273.931} C_VEL
LIN {X 0,Y 495.756,Z 396.23,A -85,B 0,C 180,E1 -6277.138,E2 -6277.138} C_VEL
LIN {X 0,Y 495.767,Z 396.227,A -85,B 0,C 180,E1 -6280.109,E2 -6280.109} C_VEL
LIN {X 0,Y 495.783,Z 396.232,A -85,B 0,C 180,E1 -6282.681,E2 -6282.681} C_VEL
LIN {X 0,Y 495.784,Z 396.224,A -85,B 0,C 180,E1 -6285.217,E2 -6285.217} C_VEL
LIN {X 0,Y 495.845,Z 396.224,A -85,B 0,C 180,E1 -6288.554,E2 -6288.554} C_VEL
LIN {X 0,Y 495.867,Z 396.214,A -85,B 0,C 180,E1 -6291.852,E2 -6291.852} C_VEL
LIN {X 0,Y 495.89,Z 396.216,A -85,B 0,C 180,E1 -6294.306,E2 -6294.306} C_VEL
LIN {X 0,Y 495.988,Z 396.198,A -85,B 0,C 180,E1 -6297.563,E2 -6297.563} C_VEL
LIN {X 0,Y 495.991,Z 396.201,A -85,B 0,C 180,E1 -6300,E2 -6300} C_VEL
LIN {X 0,Y 495.987,Z 396.205,A -85,B 0,C 180,E1 -6302.436,E2 -6302.436} C_VEL
LIN {X 0,Y 495.89,Z 396.211,A -85,B 0,C 180,E1 -6305.693,E2 -6305.693} C_VEL
LIN {X 0,Y 495.866,Z 396.22,A -85,B 0,C 180,E1 -6308.148,E2 -6308.148} C_VEL
LIN {X 0,Y 495.844,Z 396.216,A -85,B 0,C 180,E1 -6311.445,E2 -6311.445} C_VEL
LIN {X 0,Y 495.783,Z 396.224,A -85,B 0,C 180,E1 -6314.783,E2 -6314.783} C_VEL
LIN {X 0,Y 495.78,Z 396.224,A -85,B 0,C 180,E1 -6317.318,E2 -6317.318} C_VEL
LIN {X 0,Y 495.764,Z 396.231,A -85,B 0,C 180,E1 -6319.89,E2 -6319.89} C_VEL
LIN {X 0,Y 495.757,Z 396.227,A -85,B 0,C 180,E1 -6322.862,E2 -6322.862} C_VEL
LIN {X 0,Y 495.792,Z 396.23,A -85,B 0,C 180,E1 -6326.067,E2 -6326.067} C_VEL
LIN {X 0,Y 495.773,Z 396.225,A -85,B 0,C 180,E1 -6328.814,E2 -6328.814} C_VEL
LIN {X 0,Y 495.752,Z 396.233,A -85,B 0,C 180,E1 -6331.726,E2 -6331.726} C_VEL
LIN {X 0,Y 495.77,Z 396.225,A -85,B 0,C 180,E1 -6334.695,E2 -6334.695} C_VEL
LIN {X 0,Y 495.726,Z 396.235,A -85,B 0,C 180,E1 -6337.561,E2 -6337.561} C_VEL
LIN {X 0,Y 495.786,Z 396.227,A -85,B 0,C 180,E1 -6340.052,E2 -6340.052} C_VEL
LIN {X 0,Y 495.757,Z 396.227,A -85,B 0,C 180,E1 -6342.879,E2 -6342.879} C_VEL
LIN {X 0,Y 495.73,Z 396.234,A -85,B 0,C 180,E1 -6346,E2 -6346} C_VEL
LIN {X 0,Y 495.762,Z 396.226,A -85,B 0,C 180,E1 -6348.705,E2 -6348.705} C_VEL
LIN {X 0,Y 495.749,Z 396.233,A -85,B 0,C 180,E1 -6351.409,E2 -6351.409} C_VEL
LIN {X 0,Y 495.752,Z 396.227,A -85,B 0,C 180,E1 -6354.463,E2 -6354.463} C_VEL
LIN {X 0,Y 495.764,Z 396.233,A -85,B 0,C 180,E1 -6357.406,E2 -6357.406} C_VEL
LIN {X 0,Y 495.761,Z 396.226,A -85,B 0,C 180,E1 -6360.254,E2 -6360.254} C_VEL
LIN {X 0,Y 495.748,Z 396.228,A -85,B 0,C 180,E1 -6360.762,E2 -6360.762} C_VEL
LIN {X 0,Y 495.092,Z 396.318,A -85,B 0,C 180,E1 -6361.441,E2 -6361.441} C_VEL
LIN {X 0,Y 492.24,Z 396.669,A -85,B 0,C 180,E1 -6362.544,E2 -6362.544} C_VEL
LIN {X 0,Y 489.833,Z 396.973,A -85,B 0,C 180,E1 -6363.432,E2 -6363.432} C_VEL
LIN {X 0,Y 488.815,Z 397.092,A -85,B 0,C 180,E1 -6364.119,E2 -6364.119} C_VEL
LIN {X 0,Y 488.742,Z 397.1,A -85,B 0,C 180,E1 -6364.351,E2 -6364.351} C_VEL
LIN {X 0,Y 488.716,Z 397.109,A -85,B 0,C 180,E1 -6367.153,E2 -6367.153} C_VEL
LIN {X 0,Y 488.724,Z 397.106,A -85,B 0,C 180,E1 -6369.811,E2 -6369.811} C_VEL
LIN {X 0,Y 488.729,Z 397.104,A -85,B 0,C 180,E1 -6372.424,E2 -6372.424} C_VEL
LIN {X 0,Y 488.758,Z 397.106,A -85,B 0,C 180,E1 -6375,E2 -6375} C_VEL
LIN {X 0,Y 488.802,Z 397.095,A -85,B 0,C 180,E1 -6378.388,E2 -6378.388} C_VEL
LIN {X 0,Y 488.814,Z 397.096,A -85,B 0,C 180,E1 -6381.734,E2 -6381.734} C_VEL
LIN {X 0,Y 488.855,Z 397.089,A -85,B 0,C 180,E1 -6384.225,E2 -6384.225} C_VEL
LIN {X 0,Y 488.959,Z 397.078,A -85,B 0,C 180,E1 -6387.529,E2 -6387.529} C_VEL
LIN {X 0,Y 488.951,Z 397.081,A -85,B 0,C 180,E1 -6390.824,E2 -6390.824} C_VEL
LIN {X 0,Y 488.959,Z 397.078,A -85,B 0,C 180,E1 -6392.472,E2 -6392.472} C_VEL
LIN {X 0,Y 488.856,Z 397.089,A -85,B 0,C 180,E1 -6395.776,E2 -6395.776} C_VEL
LIN {X 0,Y 488.815,Z 397.095,A -85,B 0,C 180,E1 -6398.266,E2 -6398.266} C_VEL
LIN {X 0,Y 488.802,Z 397.095,A -85,B 0,C 180,E1 -6401.613,E2 -6401.613} C_VEL
LIN {X 0,Y 488.758,Z 397.106,A -85,B 0,C 180,E1 -6405,E2 -6405} C_VEL
LIN {X 0,Y 488.751,Z 397.105,A -85,B 0,C 180,E1 -6408.442,E2 -6408.442} C_VEL
LIN {X 0,Y 488.704,Z 397.108,A -85,B 0,C 180,E1 -6411.071,E2 -6411.071} C_VEL
LIN {X 0,Y 488.69,Z 397.107,A -85,B 0,C 180,E1 -6413.745,E2 -6413.745} C_VEL
LIN {X 0,Y 488.795,Z 397.097,A -85,B 0,C 180,E1 -6416.945,E2 -6416.945} C_VEL
LIN {X 0,Y 488.706,Z 397.111,A -85,B 0,C 180,E1 -6420.363,E2 -6420.363} C_VEL
LIN {X 0,Y 488.731,Z 397.102,A -85,B 0,C 180,E1 -6423.485,E2 -6423.485} C_VEL
LIN {X 0,Y 488.685,Z 397.115,A -85,B 0,C 180,E1 -6426.356,E2 -6426.356} C_VEL
LIN {X 0,Y 488.738,Z 397.101,A -85,B 0,C 180,E1 -6429.25,E2 -6429.25} C_VEL
LIN {X 0,Y 488.727,Z 397.108,A -85,B 0,C 180,E1 -6432.521,E2 -6432.521} C_VEL
LIN {X 0,Y 488.707,Z 397.105,A -85,B 0,C 180,E1 -6435.199,E2 -6435.199} C_VEL
LIN {X 0,Y 488.703,Z 397.112,A -85,B 0,C 180,E1 -6438.4,E2 -6438.4} C_VEL
LIN {X 0,Y 488.699,Z 397.106,A -85,B 0,C 180,E1 -6440.947,E2 -6440.947} C_VEL
LIN {X 0,Y 488.68,Z 397.112,A -85,B 0,C 180,E1 -6443.869,E2 -6443.869} C_VEL
LIN {X 0,Y 488.734,Z 397.102,A -85,B 0,C 180,E1 -6446.878,E2 -6446.878} C_VEL
LIN {X 0,Y 488.729,Z 397.106,A -85,B 0,C 180,E1 -6449.782,E2 -6449.782} C_VEL
LIN {X 0,Y 488.787,Z 397.095,A -85,B 0,C 180,E1 -6453.057,E2 -6453.057} C_VEL
LIN {X 0,Y 488.689,Z 397.112,A -85,B 0,C 180,E1 -6456.255,E2 -6456.255} C_VEL
LIN {X 0,Y 488.741,Z 397.101,A -85,B 0,C 180,E1 -6459.176,E2 -6459.176} C_VEL
LIN {X 0,Y 488.73,Z 397.104,A -85,B 0,C 180,E1 -6462.424,E2 -6462.424} C_VEL
LIN {X 0,Y 488.757,Z 397.099,A -85,B 0,C 180,E1 -6465,E2 -6465} C_VEL
LIN {X 0,Y 488.801,Z 397.094,A -85,B 0,C 180,E1 -6468.388,E2 -6468.388} C_VEL
LIN {X 0,Y 488.814,Z 397.1,A -85,B 0,C 180,E1 -6471.734,E2 -6471.734} C_VEL
LIN {X 0,Y 488.851,Z 397.089,A -85,B 0,C 180,E1 -6474.225,E2 -6474.225} C_VEL
LIN {X 0,Y 488.957,Z 397.08,A -85,B 0,C 180,E1 -6477.529,E2 -6477.529} C_VEL
LIN {X 0,Y 488.951,Z 397.075,A -85,B 0,C 180,E1 -6480.824,E2 -6480.824} C_VEL
LIN {X 0,Y 488.958,Z 397.073,A -85,B 0,C 180,E1 -6482.472,E2 -6482.472} C_VEL
LIN {X 0,Y 488.852,Z 397.092,A -85,B 0,C 180,E1 -6485.776,E2 -6485.776} C_VEL
LIN {X 0,Y 488.814,Z 397.092,A -85,B 0,C 180,E1 -6488.267,E2 -6488.267} C_VEL
LIN {X 0,Y 488.802,Z 397.099,A -85,B 0,C 180,E1 -6491.613,E2 -6491.613} C_VEL
LIN {X 0,Y 488.759,Z 397.102,A -85,B 0,C 180,E1 -6495.001,E2 -6495.001} C_VEL
LIN {X 0,Y 488.752,Z 397.099,A -85,B 0,C 180,E1 -6498.443,E2 -6498.443} C_VEL
LIN {X 0,Y 488.704,Z 397.11,A -85,B 0,C 180,E1 -6501.071,E2 -6501.071} C_VEL
LIN {X 0,Y 488.69,Z 397.109,A -85,B 0,C 180,E1 -6503.746,E2 -6503.746} C_VEL
LIN {X 0,Y 488.79,Z 397.099,A -85,B 0,C 180,E1 -6506.944,E2 -6506.944} C_VEL
LIN {X 0,Y 488.709,Z 397.105,A -85,B 0,C 180,E1 -6510.364,E2 -6510.364} C_VEL
LIN {X 0,Y 488.735,Z 397.106,A -85,B 0,C 180,E1 -6513.485,E2 -6513.485} C_VEL
LIN {X 0,Y 488.688,Z 397.11,A -85,B 0,C 180,E1 -6516.356,E2 -6516.356} C_VEL
LIN {X 0,Y 488.701,Z 397.113,A -85,B 0,C 180,E1 -6519.255,E2 -6519.255} C_VEL
LIN {X 0,Y 488.708,Z 397.112,A -85,B 0,C 180,E1 -6521.601,E2 -6521.601} C_VEL
LIN {X 0,Y 488.71,Z 397.112,A -85,B 0,C 180,E1 -6522.827,E2 -6522.827} C_VEL
LIN {X 0,Y 488.833,Z 397.978,A -85,B 0,C 180,E1 -6524.041,E2 -6524.041} C_VEL
LIN {X 0,Y 489.425,Z 401.874,A -85,B 0,C 180,E1 -6527.084,E2 -6527.084} C_VEL
LIN {X 0,Y 489.595,Z 404.071,A -85,B 0,C 180,E1 -6528.676,E2 -6528.676} C_VEL
LIN {X 0,Y 489.492,Z 407.264,A -85,B 0,C 180,E1 -6530.834,E2 -6530.834} C_VEL
LIN {X 0,Y 489.169,Z 412.144,A -85,B 0,C 180,E1 -6533.91,E2 -6533.91} C_VEL
LIN {X 0,Y 488.937,Z 417.19,A -85,B 0,C 180,E1 -6536.893,E2 -6536.893} C_VEL
LIN {X 0,Y 488.748,Z 422.343,A -85,B 0,C 180,E1 -6539.783,E2 -6539.783} C_VEL
LIN {X 0,Y 488.55,Z 428.583,A -85,B 0,C 180,E1 -6543.113,E2 -6543.113} C_VEL
LIN {X 0,Y 488.381,Z 434.704,A -85,B 0,C 180,E1 -6546.239,E2 -6546.239} C_VEL
LIN {X 0,Y 488.326,Z 441.036,A -85,B 0,C 180,E1 -6549.307,E2 -6549.307} C_VEL
LIN {X 0,Y 488.123,Z 447.46,A -85,B 0,C 180,E1 -6552.401,E2 -6552.401} C_VEL
LIN {X 0,Y 488.061,Z 453.523,A -85,B 0,C 180,E1 -6555.298,E2 -6555.298} C_VEL
LIN {X 0,Y 490.22,Z 465.688,A -85,B 0,C 180,E1 -6555.682,E2 -6555.682} C_VEL
LIN {X 0,Y 490.806,Z 470.447,A -85,B 0,C 180,E1 -6555.858,E2 -6555.858} C_VEL
LIN {X 0,Y 490.509,Z 482.362,A -85,B 0,C 180,E1 -6556.378,E2 -6556.378} C_VEL
LIN {X 0,Y 490.158,Z 492.234,A -85,B 0,C 180,E1 -6556.932,E2 -6556.932} C_VEL
LIN {X 0,Y 489.833,Z 501.459,A -85,B 0,C 180,E1 -6557.572,E2 -6557.572} C_VEL
LIN {X 0,Y 489.5,Z 510.16,A -85,B 0,C 180,E1 -6558.299,E2 -6558.299} C_VEL
LIN {X 0,Y 489.174,Z 517.529,A -85,B 0,C 180,E1 -6559.026,E2 -6559.026} C_VEL
LIN {X 0,Y 488.891,Z 524.72,A -85,B 0,C 180,E1 -6559.857,E2 -6559.857} C_VEL
LIN {X 0,Y 488.594,Z 532.266,A -85,B 0,C 180,E1 -6560.896,E2 -6560.896} C_VEL
LIN {X 0,Y 488.362,Z 538.554,A -85,B 0,C 180,E1 -6561.934,E2 -6561.934} C_VEL
LIN {X 0,Y 488.185,Z 543.788,A -85,B 0,C 180,E1 -6562.971,E2 -6562.971} C_VEL
LIN {X 0,Y 488.099,Z 548.885,A -85,B 0,C 180,E1 -6564.215,E2 -6564.215} C_VEL
LIN {X 0,Y 487.937,Z 552.843,A -85,B 0,C 180,E1 -6565.456,E2 -6565.456} C_VEL
LIN {X 0,Y 487.967,Z 555.766,A -85,B 0,C 180,E1 -6566.697,E2 -6566.697} C_VEL
LIN {X 0,Y 487.889,Z 558.193,A -85,B 0,C 180,E1 -6568.349,E2 -6568.349} C_VEL
LIN {X 0,Y 487.834,Z 558.777,A -85,B 0,C 180,E1 -6569.174,E2 -6569.174} C_VEL
LIN {X 0,Y 487.834,Z 558.777,A -85,B 0,C 180,E1 -6570.825,E2 -6570.825} C_VEL
LIN {X 0,Y 487.889,Z 558.193,A -85,B 0,C 180,E1 -6571.651,E2 -6571.651} C_VEL
LIN {X 0,Y 487.967,Z 555.767,A -85,B 0,C 180,E1 -6573.302,E2 -6573.302} C_VEL
LIN {X 0,Y 487.937,Z 552.844,A -85,B 0,C 180,E1 -6574.543,E2 -6574.543} C_VEL
LIN {X 0,Y 488.101,Z 548.887,A -85,B 0,C 180,E1 -6575.784,E2 -6575.784} C_VEL
LIN {X 0,Y 488.185,Z 543.79,A -85,B 0,C 180,E1 -6577.028,E2 -6577.028} C_VEL
LIN {X 0,Y 488.361,Z 538.556,A -85,B 0,C 180,E1 -6578.066,E2 -6578.066} C_VEL
LIN {X 0,Y 488.593,Z 532.268,A -85,B 0,C 180,E1 -6579.104,E2 -6579.104} C_VEL
LIN {X 0,Y 488.891,Z 524.723,A -85,B 0,C 180,E1 -6580.142,E2 -6580.142} C_VEL
LIN {X 0,Y 489.269,Z 515.617,A -85,B 0,C 180,E1 -6581.181,E2 -6581.181} C_VEL
LIN {X 0,Y 489.763,Z 504.161,A -85,B 0,C 180,E1 -6582.219,E2 -6582.219} C_VEL
LIN {X 0,Y 490.026,Z 495.332,A -85,B 0,C 180,E1 -6582.871,E2 -6582.871} C_VEL
LIN {X 0,Y 490.327,Z 485.386,A -85,B 0,C 180,E1 -6583.468,E2 -6583.468} C_VEL
LIN {X 0,Y 490.663,Z 475.602,A -85,B 0,C 180,E1 -6583.934,E2 -6583.934} C_VEL
LIN {X 0,Y 490.653,Z 468.3,A -85,B 0,C 180,E1 -6584.225,E2 -6584.225} C_VEL
LIN {X 0,Y 488.467,Z 455.708,A -85,B 0,C 180,E1 -6584.639,E2 -6584.639} C_VEL
LIN {X 0,Y 488.079,Z 453.524,A -85,B 0,C 180,E1 -6584.701,E2 -6584.701} C_VEL
LIN {X 0,Y 488.164,Z 445.664,A -85,B 0,C 180,E1 -6588.465,E2 -6588.465} C_VEL
LIN {X 0,Y 488.3,Z 440.215,A -85,B 0,C 180,E1 -6591.089,E2 -6591.089} C_VEL
LIN {X 0,Y 488.38,Z 434.705,A -85,B 0,C 180,E1 -6593.761,E2 -6593.761} C_VEL
LIN {X 0,Y 488.548,Z 428.583,A -85,B 0,C 180,E1 -6596.886,E2 -6596.886} C_VEL
LIN {X 0,Y 488.746,Z 422.333,A -85,B 0,C 180,E1 -6600.217,E2 -6600.217} C_VEL
LIN {X 0,Y 488.968,Z 416.453,A -85,B 0,C 180,E1 -6603.525,E2 -6603.525} C_VEL
LIN {X 0,Y 489.188,Z 411.579,A -85,B 0,C 180,E1 -6606.434,E2 -6606.434} C_VEL
LIN {X 0,Y 489.465,Z 407.239,A -85,B 0,C 180,E1 -6609.18,E2 -6609.18} C_VEL
LIN {X 0,Y 489.582,Z 403.503,A -85,B 0,C 180,E1 -6611.714,E2 -6611.714} C_VEL
LIN {X 0,Y 489.212,Z 400.313,A -85,B 0,C 180,E1 -6614.085,E2 -6614.085} C_VEL
LIN {X 0,Y 488.76,Z 397.501,A -85,B 0,C 180,E1 -6616.353,E2 -6616.353} C_VEL
LIN {X 0,Y 488.689,Z 397.113,A -85,B 0,C 180,E1 -6617.474,E2 -6617.474} C_VEL
LIN {X 0,Y 488.73,Z 397.107,A -85,B 0,C 180,E1 -6619.676,E2 -6619.676} C_VEL
LIN {X 0,Y 488.68,Z 397.117,A -85,B 0,C 180,E1 -6622.841,E2 -6622.841} C_VEL
LIN {X 0,Y 488.731,Z 397.102,A -85,B 0,C 180,E1 -6625.887,E2 -6625.887} C_VEL
LIN {X 0,Y 488.714,Z 397.112,A -85,B 0,C 180,E1 -6628.821,E2 -6628.821} C_VEL
LIN {X 0,Y 488.742,Z 397.1,A -85,B 0,C 180,E1 -6631.671,E2 -6631.671} C_VEL
LIN {X 0,Y 488.743,Z 397.104,A -85,B 0,C 180,E1 -6634.444,E2 -6634.444} C_VEL
LIN {X 0,Y 488.719,Z 397.106,A -85,B 0,C 180,E1 -6637.153,E2 -6637.153} C_VEL
LIN {X 0,Y 488.72,Z 397.103,A -85,B 0,C 180,E1 -6639.81,E2 -6639.81} C_VEL
LIN {X 0,Y 488.73,Z 397.107,A -85,B 0,C 180,E1 -6642.423,E2 -6642.423} C_VEL
LIN {X 0,Y 488.756,Z 397.102,A -85,B 0,C 180,E1 -6644.999,E2 -6644.999} C_VEL
LIN {X 0,Y 488.799,Z 397.099,A -85,B 0,C 180,E1 -6648.387,E2 -6648.387} C_VEL
LIN {X 0,Y 488.811,Z 397.092,A -85,B 0,C 180,E1 -6651.733,E2 -6651.733} C_VEL
LIN {X 0,Y 488.85,Z 397.092,A -85,B 0,C 180,E1 -6654.224,E2 -6654.224} C_VEL
LIN {X 0,Y 488.955,Z 397.074,A -85,B 0,C 180,E1 -6657.528,E2 -6657.528} C_VEL
LIN {X 0,Y 488.948,Z 397.077,A -85,B 0,C 180,E1 -6660.823,E2 -6660.823} C_VEL
LIN {X 0,Y 488.955,Z 397.081,A -85,B 0,C 180,E1 -6662.471,E2 -6662.471} C_VEL
LIN {X 0,Y 488.849,Z 397.089,A -85,B 0,C 180,E1 -6665.775,E2 -6665.775} C_VEL
LIN {X 0,Y 488.811,Z 397.101,A -85,B 0,C 180,E1 -6668.266,E2 -6668.266} C_VEL
LIN {X 0,Y 488.798,Z 397.095,A -85,B 0,C 180,E1 -6671.612,E2 -6671.612} C_VEL
LIN {X 0,Y 488.754,Z 397.099,A -85,B 0,C 180,E1 -6675,E2 -6675} C_VEL
LIN {X 0,Y 488.747,Z 397.104,A -85,B 0,C 180,E1 -6678.442,E2 -6678.442} C_VEL
LIN {X 0,Y 488.699,Z 397.106,A -85,B 0,C 180,E1 -6681.071,E2 -6681.071} C_VEL
LIN {X 0,Y 488.686,Z 397.112,A -85,B 0,C 180,E1 -6683.745,E2 -6683.745} C_VEL
LIN {X 0,Y 488.791,Z 397.094,A -85,B 0,C 180,E1 -6686.945,E2 -6686.945} C_VEL
LIN {X 0,Y 488.711,Z 397.107,A -85,B 0,C 180,E1 -6690.365,E2 -6690.365} C_VEL
LIN {X 0,Y 488.729,Z 397.105,A -85,B 0,C 180,E1 -6693.485,E2 -6693.485} C_VEL
LIN {X 0,Y 488.682,Z 397.11,A -85,B 0,C 180,E1 -6696.356,E2 -6696.356} C_VEL
LIN {X 0,Y 488.741,Z 397.102,A -85,B 0,C 180,E1 -6699.25,E2 -6699.25} C_VEL
LIN {X 0,Y 488.728,Z 397.102,A -85,B 0,C 180,E1 -6702.521,E2 -6702.521} C_VEL
LIN {X 0,Y 488.695,Z 397.11,A -85,B 0,C 180,E1 -6705.976,E2 -6705.976} C_VEL
LIN {X 0,Y 488.718,Z 397.103,A -85,B 0,C 180,E1 -6708.586,E2 -6708.586} C_VEL
LIN {X 0,Y 488.734,Z 397.102,A -85,B 0,C 180,E1 -6710.942,E2 -6710.942} C_VEL
LIN {X 0,Y 488.68,Z 397.112,A -85,B 0,C 180,E1 -6713.869,E2 -6713.869} C_VEL
LIN {X 0,Y 488.734,Z 397.102,A -85,B 0,C 180,E1 -6716.878,E2 -6716.878} C_VEL
LIN {X 0,Y 488.718,Z 397.107,A -85,B 0,C 180,E1 -6719.781,E2 -6719.781} C_VEL
LIN {X 0,Y 488.794,Z 397.097,A -85,B 0,C 180,E1 -6723.055,E2 -6723.055} C_VEL
LIN {X 0,Y 488.742,Z 397.1,A -85,B 0,C 180,E1 -6724.351,E2 -6724.351} C_VEL
LIN {X 0,Y 488.094,Z 397.186,A -85,B 0,C 180,E1 -6725.039,E2 -6725.039} C_VEL
LIN {X 0,Y 485.224,Z 397.542,A -85,B 0,C 180,E1 -6726.155,E2 -6726.155} C_VEL
LIN {X 0,Y 482.778,Z 397.848,A -85,B 0,C 180,E1 -6727.055,E2 -6727.055} C_VEL
LIN {X 0,Y 481.721,Z 397.979,A -85,B 0,C 180,E1 -6727.75,E2 -6727.75} C_VEL
LIN {X 0,Y 481.632,Z 397.987,A -85,B 0,C 180,E1 -6727.986,E2 -6727.986} C_VEL
LIN {X 0,Y 481.703,Z 397.977,A -85,B 0,C 180,E1 -6730.393,E2 -6730.393} C_VEL
LIN {X 0,Y 481.687,Z 397.987,A -85,B 0,C 180,E1 -6733.034,E2 -6733.034} C_VEL
LIN {X 0,Y 481.686,Z 397.985,A -85,B 0,C 180,E1 -6735.639,E2 -6735.639} C_VEL
LIN {X 0,Y 481.747,Z 397.973,A -85,B 0,C 180,E1 -6738.215,E2 -6738.215} C_VEL
LIN {X 0,Y 481.76,Z 397.975,A -85,B 0,C 180,E1 -6741.612,E2 -6741.612} C_VEL
LIN {X 0,Y 481.816,Z 397.966,A -85,B 0,C 180,E1 -6744.14,E2 -6744.14} C_VEL
LIN {X 0,Y 481.926,Z 397.955,A -85,B 0,C 180,E1 -6747.493,E2 -6747.493} C_VEL
LIN {X 0,Y 481.902,Z 397.959,A -85,B 0,C 180,E1 -6750.836,E2 -6750.836} C_VEL
LIN {X 0,Y 481.926,Z 397.955,A -85,B 0,C 180,E1 -6752.508,E2 -6752.508} C_VEL
LIN {X 0,Y 481.816,Z 397.966,A -85,B 0,C 180,E1 -6755.861,E2 -6755.861} C_VEL
LIN {X 0,Y 481.76,Z 397.975,A -85,B 0,C 180,E1 -6758.388,E2 -6758.388} C_VEL
LIN {X 0,Y 481.748,Z 397.973,A -85,B 0,C 180,E1 -6761.785,E2 -6761.785} C_VEL
LIN {X 0,Y 481.739,Z 397.978,A -85,B 0,C 180,E1 -6765.224,E2 -6765.224} C_VEL
LIN {X 0,Y 481.709,Z 397.985,A -85,B 0,C 180,E1 -6768.722,E2 -6768.722} C_VEL
LIN {X 0,Y 481.644,Z 397.985,A -85,B 0,C 180,E1 -6771.395,E2 -6771.395} C_VEL
LIN {X 0,Y 481.674,Z 397.983,A -85,B 0,C 180,E1 -6774.113,E2 -6774.113} C_VEL
LIN {X 0,Y 481.748,Z 397.973,A -85,B 0,C 180,E1 -6777.141,E2 -6777.141} C_VEL
LIN {X 0,Y 481.675,Z 397.981,A -85,B 0,C 180,E1 -6779.741,E2 -6779.741} C_VEL
LIN {X 0,Y 481.669,Z 397.987,A -85,B 0,C 180,E1 -6782.674,E2 -6782.674} C_VEL
LIN {X 0,Y 481.639,Z 397.986,A -85,B 0,C 180,E1 -6785.709,E2 -6785.709} C_VEL
LIN {X 0,Y 481.71,Z 397.976,A -85,B 0,C 180,E1 -6789.354,E2 -6789.354} C_VEL
LIN {X 0,Y 481.669,Z 397.987,A -85,B 0,C 180,E1 -6792.158,E2 -6792.158} C_VEL
LIN {X 0,Y 481.655,Z 397.99,A -85,B 0,C 180,E1 -6794.457,E2 -6794.457} C_VEL
LIN {X 0,Y 481.642,Z 397.988,A -85,B 0,C 180,E1 -6797.839,E2 -6797.839} C_VEL
LIN {X 0,Y 481.675,Z 397.983,A -85,B 0,C 180,E1 -6800.651,E2 -6800.651} C_VEL
LIN {X 0,Y 481.626,Z 397.987,A -85,B 0,C 180,E1 -6803.376,E2 -6803.376} C_VEL
LIN {X 0,Y 481.704,Z 397.983,A -85,B 0,C 180,E1 -6806.33,E2 -6806.33} C_VEL
LIN {X 0,Y 481.653,Z 397.984,A -85,B 0,C 180,E1 -6809.416,E2 -6809.416} C_VEL
LIN {X 0,Y 481.696,Z 397.985,A -85,B 0,C 180,E1 -6812.168,E2 -6812.168} C_VEL
LIN {X 0,Y 481.713,Z 397.976,A -85,B 0,C 180,E1 -6814.97,E2 -6814.97} C_VEL
LIN {X 0,Y 481.648,Z 397.989,A -85,B 0,C 180,E1 -6817.705,E2 -6817.705} C_VEL
LIN {X 0,Y 481.701,Z 397.98,A -85,B 0,C 180,E1 -6820.393,E2 -6820.393} C_VEL
LIN {X 0,Y 481.687,Z 397.979,A -85,B 0,C 180,E1 -6823.034,E2 -6823.034} C_VEL
LIN {X 0,Y 481.686,Z 397.985,A -85,B 0,C 180,E1 -6825.639,E2 -6825.639} C_VEL
LIN {X 0,Y 481.746,Z 397.975,A -85,B 0,C 180,E1 -6828.215,E2 -6828.215} C_VEL
LIN {X 0,Y 481.759,Z 397.977,A -85,B 0,C 180,E1 -6831.612,E2 -6831.612} C_VEL
LIN {X 0,Y 481.812,Z 397.966,A -85,B 0,C 180,E1 -6834.14,E2 -6834.14} C_VEL
LIN {X 0,Y 481.924,Z 397.956,A -85,B 0,C 180,E1 -6837.493,E2 -6837.493} C_VEL
LIN {X 0,Y 481.902,Z 397.953,A -85,B 0,C 180,E1 -6840.836,E2 -6840.836} C_VEL
LIN {X 0,Y 481.925,Z 397.95,A -85,B 0,C 180,E1 -6842.508,E2 -6842.508} C_VEL
LIN {X 0,Y 481.813,Z 397.967,A -85,B 0,C 180,E1 -6845.861,E2 -6845.861} C_VEL
LIN {X 0,Y 481.76,Z 397.97,A -85,B 0,C 180,E1 -6848.389,E2 -6848.389} C_VEL
LIN {X 0,Y 481.747,Z 397.975,A -85,B 0,C 180,E1 -6851.785,E2 -6851.785} C_VEL
LIN {X 0,Y 481.74,Z 397.979,A -85,B 0,C 180,E1 -6855.225,E2 -6855.225} C_VEL
LIN {X 0,Y 481.71,Z 397.978,A -85,B 0,C 180,E1 -6858.722,E2 -6858.722} C_VEL
LIN {X 0,Y 481.644,Z 397.991,A -85,B 0,C 180,E1 -6861.395,E2 -6861.395} C_VEL
LIN {X 0,Y 481.675,Z 397.981,A -85,B 0,C 180,E1 -6864.114,E2 -6864.114} C_VEL
LIN {X 0,Y 481.745,Z 397.98,A -85,B 0,C 180,E1 -6867.14,E2 -6867.14} C_VEL
LIN {X 0,Y 481.677,Z 397.982,A -85,B 0,C 180,E1 -6869.742,E2 -6869.742} C_VEL
LIN {X 0,Y 481.672,Z 397.984,A -85,B 0,C 180,E1 -6872.675,E2 -6872.675} C_VEL
LIN {X 0,Y 481.642,Z 397.988,A -85,B 0,C 180,E1 -6875.71,E2 -6875.71} C_VEL
LIN {X 0,Y 481.671,Z 397.989,A -85,B 0,C 180,E1 -6878.86,E2 -6878.86} C_VEL
LIN {X 0,Y 481.653,Z 397.99,A -85,B 0,C 180,E1 -6881.914,E2 -6881.914} C_VEL
LIN {X 0,Y 481.72,Z 398.334,A -85,B 0,C 180,E1 -6883.291,E2 -6883.291} C_VEL
LIN {X 0,Y 482.163,Z 401.142,A -85,B 0,C 180,E1 -6885.602,E2 -6885.602} C_VEL
LIN {X 0,Y 482.541,Z 404.266,A -85,B 0,C 180,E1 -6887.97,E2 -6887.97} C_VEL
LIN {X 0,Y 482.486,Z 407.934,A -85,B 0,C 180,E1 -6890.535,E2 -6890.535} C_VEL
LIN {X 0,Y 482.194,Z 412.217,A -85,B 0,C 180,E1 -6893.304,E2 -6893.304} C_VEL
LIN {X 0,Y 481.947,Z 417.218,A -85,B 0,C 180,E1 -6896.349,E2 -6896.349} C_VEL
LIN {X 0,Y 481.708,Z 422.553,A -85,B 0,C 180,E1 -6899.407,E2 -6899.407} C_VEL
LIN {X 0,Y 481.523,Z 427.575,A -85,B 0,C 180,E1 -6902.157,E2 -6902.157} C_VEL
LIN {X 0,Y 481.38,Z 432.853,A -85,B 0,C 180,E1 -6904.951,E2 -6904.951} C_VEL
LIN {X 0,Y 481.241,Z 438.272,A -85,B 0,C 180,E1 -6907.685,E2 -6907.685} C_VEL
LIN {X 0,Y 481.14,Z 443.773,A -85,B 0,C 180,E1 -6910.369,E2 -6910.369} C_VEL
LIN {X 0,Y 480.988,Z 449.257,A -85,B 0,C 180,E1 -6913.008,E2 -6913.008} C_VEL
LIN {X 0,Y 481.022,Z 453.523,A -85,B 0,C 180,E1 -6915.078,E2 -6915.078} C_VEL
LIN {X 0,Y 483.165,Z 465.672,A -85,B 0,C 180,E1 -6915.468,E2 -6915.468} C_VEL
LIN {X 0,Y 483.882,Z 471.725,A -85,B 0,C 180,E1 -6915.705,E2 -6915.705} C_VEL
LIN {X 0,Y 483.61,Z 482.353,A -85,B 0,C 180,E1 -6916.18,E2 -6916.18} C_VEL
LIN {X 0,Y 483.207,Z 492.801,A -85,B 0,C 180,E1 -6916.779,E2 -6916.779} C_VEL
LIN {X 0,Y 482.872,Z 501.451,A -85,B 0,C 180,E1 -6917.39,E2 -6917.39} C_VEL
LIN {X 0,Y 482.531,Z 510.154,A -85,B 0,C 180,E1 -6918.128,E2 -6918.128} C_VEL
LIN {X 0,Y 482.185,Z 517.524,A -85,B 0,C 180,E1 -6918.865,E2 -6918.865} C_VEL
LIN {X 0,Y 481.886,Z 524.716,A -85,B 0,C 180,E1 -6919.708,E2 -6919.708} C_VEL
LIN {X 0,Y 481.577,Z 532.262,A -85,B 0,C 180,E1 -6920.762,E2 -6920.762} C_VEL
LIN {X 0,Y 481.325,Z 538.55,A -85,B 0,C 180,E1 -6921.815,E2 -6921.815} C_VEL
LIN {X 0,Y 481.101,Z 543.783,A -85,B 0,C 180,E1 -6922.867,E2 -6922.867} C_VEL
LIN {X 0,Y 480.989,Z 547.531,A -85,B 0,C 180,E1 -6923.761,E2 -6923.761} C_VEL
LIN {X 0,Y 480.906,Z 551.631,A -85,B 0,C 180,E1 -6924.969,E2 -6924.969} C_VEL
LIN {X 0,Y 480.847,Z 553.974,A -85,B 0,C 180,E1 -6925.809,E2 -6925.809} C_VEL
LIN {X 0,Y 480.892,Z 555.763,A -85,B 0,C 180,E1 -6926.649,E2 -6926.649} C_VEL
LIN {X 0,Y 480.79,Z 558.19,A -85,B 0,C 180,E1 -6928.325,E2 -6928.325} C_VEL
LIN {X 0,Y 480.76,Z 558.773,A -85,B 0,C 180,E1 -6929.162,E2 -6929.162} C_VEL
LIN {X 0,Y 480.76,Z 558.773,A -85,B 0,C 180,E1 -6930.837,E2 -6930.837} C_VEL
LIN {X 0,Y 480.79,Z 558.19,A -85,B 0,C 180,E1 -6931.675,E2 -6931.675} C_VEL
LIN {X 0,Y 480.892,Z 555.764,A -85,B 0,C 180,E1 -6933.351,E2 -6933.351} C_VEL
LIN {X 0,Y 480.853,Z 552.84,A -85,B 0,C 180,E1 -6934.611,E2 -6934.611} C_VEL
LIN {X 0,Y 481.019,Z 548.882,A -85,B 0,C 180,E1 -6935.87,E2 -6935.87} C_VEL
LIN {X 0,Y 481.061,Z 545.686,A -85,B 0,C 180,E1 -6936.712,E2 -6936.712} C_VEL
LIN {X 0,Y 481.249,Z 539.702,A -85,B 0,C 180,E1 -6937.974,E2 -6937.974} C_VEL
LIN {X 0,Y 481.524,Z 533.634,A -85,B 0,C 180,E1 -6939.027,E2 -6939.027} C_VEL
LIN {X 0,Y 481.831,Z 526.339,A -85,B 0,C 180,E1 -6940.08,E2 -6940.08} C_VEL
LIN {X 0,Y 482.084,Z 519.44,A -85,B 0,C 180,E1 -6940.924,E2 -6940.924} C_VEL
LIN {X 0,Y 482.498,Z 511.289,A -85,B 0,C 180,E1 -6941.766,E2 -6941.766} C_VEL
LIN {X 0,Y 482.832,Z 502.804,A -85,B 0,C 180,E1 -6942.504,E2 -6942.504} C_VEL
LIN {X 0,Y 483.117,Z 494.598,A -85,B 0,C 180,E1 -6943.106,E2 -6943.106} C_VEL
LIN {X 0,Y 483.464,Z 484.371,A -85,B 0,C 180,E1 -6943.717,E2 -6943.717} C_VEL
LIN {X 0,Y 483.819,Z 474.306,A -85,B 0,C 180,E1 -6944.189,E2 -6944.189} C_VEL
LIN {X 0,Y 483.605,Z 468.295,A -85,B 0,C 180,E1 -6944.437,E2 -6944.437} C_VEL
LIN {X 0,Y 481.442,Z 455.843,A -85,B 0,C 180,E1 -6944.855,E2 -6944.855} C_VEL
LIN {X 0,Y 481.041,Z 453.524,A -85,B 0,C 180,E1 -6944.921,E2 -6944.921} C_VEL
LIN {X 0,Y 481.103,Z 445.605,A -85,B 0,C 180,E1 -6948.746,E2 -6948.746} C_VEL
LIN {X 0,Y 481.232,Z 440.109,A -85,B 0,C 180,E1 -6951.414,E2 -6951.414} C_VEL
LIN {X 0,Y 481.343,Z 434.608,A -85,B 0,C 180,E1 -6954.13,E2 -6954.13} C_VEL
LIN {X 0,Y 481.507,Z 428.995,A -85,B 0,C 180,E1 -6957.082,E2 -6957.082} C_VEL
LIN {X 0,Y 481.623,Z 424.045,A -85,B 0,C 180,E1 -6959.744,E2 -6959.744} C_VEL
LIN {X 0,Y 481.855,Z 418.907,A -85,B 0,C 180,E1 -6962.659,E2 -6962.659} C_VEL
LIN {X 0,Y 482.097,Z 413.843,A -85,B 0,C 180,E1 -6965.669,E2 -6965.669} C_VEL
LIN {X 0,Y 482.423,Z 408.954,A -85,B 0,C 180,E1 -6968.786,E2 -6968.786} C_VEL
LIN {X 0,Y 482.556,Z 405.754,A -85,B 0,C 180,E1 -6970.948,E2 -6970.948} C_VEL
LIN {X 0,Y 482.362,Z 402.626,A -85,B 0,C 180,E1 -6973.239,E2 -6973.239} C_VEL
LIN {X 0,Y 481.913,Z 399.647,A -85,B 0,C 180,E1 -6975.609,E2 -6975.609} C_VEL
LIN {X 0,Y 481.682,Z 398.164,A -85,B 0,C 180,E1 -6976.846,E2 -6976.846} C_VEL
LIN {X 0,Y 481.674,Z 397.986,A -85,B 0,C 180,E1 -6980.059,E2 -6980.059} C_VEL
LIN {X 0,Y 481.627,Z 397.995,A -85,B 0,C 180,E1 -6983.253,E2 -6983.253} C_VEL
LIN {X 0,Y 481.706,Z 397.978,A -85,B 0,C 180,E1 -6986.329,E2 -6986.329} C_VEL
LIN {X 0,Y 481.661,Z 397.984,A -85,B 0,C 180,E1 -6989.414,E2 -6989.414} C_VEL
LIN {X 0,Y 481.697,Z 397.979,A -85,B 0,C 180,E1 -6992.167,E2 -6992.167} C_VEL
LIN {X 0,Y 481.713,Z 397.982,A -85,B 0,C 180,E1 -6994.969,E2 -6994.969} C_VEL
LIN {X 0,Y 481.645,Z 397.984,A -85,B 0,C 180,E1 -6997.704,E2 -6997.704} C_VEL
LIN {X 0,Y 481.7,Z 397.982,A -85,B 0,C 180,E1 -7000.392,E2 -7000.392} C_VEL
LIN {X 0,Y 481.687,Z 397.983,A -85,B 0,C 180,E1 -7003.033,E2 -7003.033} C_VEL
LIN {X 0,Y 481.684,Z 397.979,A -85,B 0,C 180,E1 -7005.638,E2 -7005.638} C_VEL
LIN {X 0,Y 481.745,Z 397.976,A -85,B 0,C 180,E1 -7008.214,E2 -7008.214} C_VEL
LIN {X 0,Y 481.757,Z 397.97,A -85,B 0,C 180,E1 -7011.611,E2 -7011.611} C_VEL
LIN {X 0,Y 481.811,Z 397.968,A -85,B 0,C 180,E1 -7014.139,E2 -7014.139} C_VEL
LIN {X 0,Y 481.922,Z 397.95,A -85,B 0,C 180,E1 -7017.492,E2 -7017.492} C_VEL
LIN {X 0,Y 481.899,Z 397.955,A -85,B 0,C 180,E1 -7020.835,E2 -7020.835} C_VEL
LIN {X 0,Y 481.922,Z 397.956,A -85,B 0,C 180,E1 -7022.507,E2 -7022.507} C_VEL
LIN {X 0,Y 481.81,Z 397.967,A -85,B 0,C 180,E1 -7025.86,E2 -7025.86} C_VEL
LIN {X 0,Y 481.756,Z 397.977,A -85,B 0,C 180,E1 -7028.388,E2 -7028.388} C_VEL
LIN {X 0,Y 481.743,Z 397.975,A -85,B 0,C 180,E1 -7031.785,E2 -7031.785} C_VEL
LIN {X 0,Y 481.735,Z 397.973,A -85,B 0,C 180,E1 -7035.224,E2 -7035.224} C_VEL
LIN {X 0,Y 481.704,Z 397.978,A -85,B 0,C 180,E1 -7038.721,E2 -7038.721} C_VEL
LIN {X 0,Y 481.639,Z 397.986,A -85,B 0,C 180,E1 -7041.394,E2 -7041.394} C_VEL
LIN {X 0,Y 481.67,Z 397.988,A -85,B 0,C 180,E1 -7044.113,E2 -7044.113} C_VEL
LIN {X 0,Y 481.744,Z 397.972,A -85,B 0,C 180,E1 -7047.14,E2 -7047.14} C_VEL
LIN {X 0,Y 481.681,Z 397.986,A -85,B 0,C 180,E1 -7049.74,E2 -7049.74} C_VEL
LIN {X 0,Y 481.666,Z 397.982,A -85,B 0,C 180,E1 -7052.674,E2 -7052.674} C_VEL
LIN {X 0,Y 481.636,Z 397.992,A -85,B 0,C 180,E1 -7055.709,E2 -7055.709} C_VEL
LIN {X 0,Y 481.712,Z 397.979,A -85,B 0,C 180,E1 -7059.355,E2 -7059.355} C_VEL
LIN {X 0,Y 481.667,Z 397.985,A -85,B 0,C 180,E1 -7062.158,E2 -7062.158} C_VEL
LIN {X 0,Y 481.653,Z 397.984,A -85,B 0,C 180,E1 -7064.457,E2 -7064.457} C_VEL
LIN {X 0,Y 481.682,Z 397.98,A -85,B 0,C 180,E1 -7066.846,E2 -7066.846} C_VEL
LIN {X 0,Y 481.683,Z 397.982,A -85,B 0,C 180,E1 -7070.061,E2 -7070.061} C_VEL
LIN {X 0,Y 481.624,Z 397.991,A -85,B 0,C 180,E1 -7073.254,E2 -7073.254} C_VEL
LIN {X 0,Y 481.703,Z 397.977,A -85,B 0,C 180,E1 -7076.33,E2 -7076.33} C_VEL
LIN {X 0,Y 481.646,Z 397.992,A -85,B 0,C 180,E1 -7079.417,E2 -7079.417} C_VEL
LIN {X 0,Y 481.697,Z 397.979,A -85,B 0,C 180,E1 -7082.169,E2 -7082.169} C_VEL
LIN {X 0,Y 481.713,Z 397.979,A -85,B 0,C 180,E1 -7084.97,E2 -7084.97} C_VEL
LIN {X 0,Y 481.632,Z 397.987,A -85,B 0,C 180,E1 -7087.986,E2 -7087.986} C_VEL
LIN {X 0,Y 480.965,Z 398.071,A -85,B 0,C 180,E1 -7088.684,E2 -7088.684} C_VEL
LIN {X 0,Y 478.137,Z 398.425,A -85,B 0,C 180,E1 -7089.818,E2 -7089.818} C_VEL
LIN {X 0,Y 475.753,Z 398.725,A -85,B 0,C 180,E1 -7090.733,E2 -7090.733} C_VEL
LIN {X 0,Y 474.732,Z 398.853,A -85,B 0,C 180,E1 -7091.438,E2 -7091.438} C_VEL
LIN {X 0,Y 474.651,Z 398.861,A -85,B 0,C 180,E1 -7091.677,E2 -7091.677} C_VEL
LIN {X 0,Y 474.696,Z 398.854,A -85,B 0,C 180,E1 -7094.545,E2 -7094.545} C_VEL
LIN {X 0,Y 474.7,Z 398.851,A -85,B 0,C 180,E1 -7098.038,E2 -7098.038} C_VEL
LIN {X 0,Y 474.725,Z 398.852,A -85,B 0,C 180,E1 -7101.487,E2 -7101.487} C_VEL
LIN {X 0,Y 474.778,Z 398.843,A -85,B 0,C 180,E1 -7104.053,E2 -7104.053} C_VEL
LIN {X 0,Y 474.892,Z 398.831,A -85,B 0,C 180,E1 -7107.456,E2 -7107.456} C_VEL
LIN {X 0,Y 474.909,Z 398.828,A -85,B 0,C 180,E1 -7110,E2 -7110} C_VEL
LIN {X 0,Y 474.892,Z 398.831,A -85,B 0,C 180,E1 -7112.545,E2 -7112.545} C_VEL
LIN {X 0,Y 474.779,Z 398.843,A -85,B 0,C 180,E1 -7115.948,E2 -7115.948} C_VEL
LIN {X 0,Y 474.725,Z 398.852,A -85,B 0,C 180,E1 -7118.514,E2 -7118.514} C_VEL
LIN {X 0,Y 474.701,Z 398.851,A -85,B 0,C 180,E1 -7121.963,E2 -7121.963} C_VEL
LIN {X 0,Y 474.696,Z 398.854,A -85,B 0,C 180,E1 -7125.456,E2 -7125.456} C_VEL
LIN {X 0,Y 474.662,Z 398.861,A -85,B 0,C 180,E1 -7129.01,E2 -7129.01} C_VEL
LIN {X 0,Y 474.586,Z 398.864,A -85,B 0,C 180,E1 -7131.729,E2 -7131.729} C_VEL
LIN {X 0,Y 474.656,Z 398.862,A -85,B 0,C 180,E1 -7134.493,E2 -7134.493} C_VEL
LIN {X 0,Y 474.695,Z 398.851,A -85,B 0,C 180,E1 -7137.339,E2 -7137.339} C_VEL
LIN {X 0,Y 474.601,Z 398.866,A -85,B 0,C 180,E1 -7140.81,E2 -7140.81} C_VEL
LIN {X 0,Y 474.634,Z 398.86,A -85,B 0,C 180,E1 -7143.984,E2 -7143.984} C_VEL
LIN {X 0,Y 474.571,Z 398.868,A -85,B 0,C 180,E1 -7146.9,E2 -7146.9} C_VEL
LIN {X 0,Y 474.646,Z 398.857,A -85,B 0,C 180,E1 -7149.651,E2 -7149.651} C_VEL
LIN {X 0,Y 474.647,Z 398.858,A -85,B 0,C 180,E1 -7152.93,E2 -7152.93} C_VEL
LIN {X 0,Y 474.604,Z 398.865,A -85,B 0,C 180,E1 -7155.895,E2 -7155.895} C_VEL
LIN {X 0,Y 474.623,Z 398.859,A -85,B 0,C 180,E1 -7159.041,E2 -7159.041} C_VEL
LIN {X 0,Y 474.606,Z 398.863,A -85,B 0,C 180,E1 -7161.704,E2 -7161.704} C_VEL
LIN {X 0,Y 474.625,Z 398.86,A -85,B 0,C 180,E1 -7164.726,E2 -7164.726} C_VEL
LIN {X 0,Y 474.633,Z 398.862,A -85,B 0,C 180,E1 -7167.788,E2 -7167.788} C_VEL
LIN {X 0,Y 474.627,Z 398.859,A -85,B 0,C 180,E1 -7170.883,E2 -7170.883} C_VEL
LIN {X 0,Y 474.655,Z 398.858,A -85,B 0,C 180,E1 -7173.629,E2 -7173.629} C_VEL
LIN {X 0,Y 474.631,Z 398.859,A -85,B 0,C 180,E1 -7176.641,E2 -7176.641} C_VEL
LIN {X 0,Y 474.65,Z 398.862,A -85,B 0,C 180,E1 -7180.09,E2 -7180.09} C_VEL
LIN {X 0,Y 474.646,Z 398.856,A -85,B 0,C 180,E1 -7182.775,E2 -7182.775} C_VEL
LIN {X 0,Y 474.644,Z 398.859,A -85,B 0,C 180,E1 -7185.421,E2 -7185.421} C_VEL
LIN {X 0,Y 474.699,Z 398.855,A -85,B 0,C 180,E1 -7188.038,E2 -7188.038} C_VEL
LIN {X 0,Y 474.724,Z 398.851,A -85,B 0,C 180,E1 -7191.487,E2 -7191.487} C_VEL
LIN {X 0,Y 474.775,Z 398.844,A -85,B 0,C 180,E1 -7194.053,E2 -7194.053} C_VEL
LIN {X 0,Y 474.89,Z 398.831,A -85,B 0,C 180,E1 -7197.456,E2 -7197.456} C_VEL
LIN {X 0,Y 474.908,Z 398.827,A -85,B 0,C 180,E1 -7200,E2 -7200} C_VEL
LIN {X 0,Y 474.891,Z 398.826,A -85,B 0,C 180,E1 -7202.545,E2 -7202.545} C_VEL
LIN {X 0,Y 474.776,Z 398.843,A -85,B 0,C 180,E1 -7205.948,E2 -7205.948} C_VEL
LIN {X 0,Y 474.725,Z 398.846,A -85,B 0,C 180,E1 -7208.514,E2 -7208.514} C_VEL
LIN {X 0,Y 474.701,Z 398.851,A -85,B 0,C 180,E1 -7211.963,E2 -7211.963} C_VEL
LIN {X 0,Y 474.697,Z 398.857,A -85,B 0,C 180,E1 -7215.456,E2 -7215.456} C_VEL
LIN {X 0,Y 474.662,Z 398.858,A -85,B 0,C 180,E1 -7219.011,E2 -7219.011} C_VEL
LIN {X 0,Y 474.586,Z 398.866,A -85,B 0,C 180,E1 -7221.729,E2 -7221.729} C_VEL
LIN {X 0,Y 474.657,Z 398.855,A -85,B 0,C 180,E1 -7224.493,E2 -7224.493} C_VEL
LIN {X 0,Y 474.679,Z 398.858,A -85,B 0,C 180,E1 -7227.335,E2 -7227.335} C_VEL
LIN {X 0,Y 474.604,Z 398.862,A -85,B 0,C 180,E1 -7230.231,E2 -7230.231} C_VEL
LIN {X 0,Y 474.642,Z 398.864,A -85,B 0,C 180,E1 -7233.221,E2 -7233.221} C_VEL
LIN {X 0,Y 474.593,Z 398.866,A -85,B 0,C 180,E1 -7236.324,E2 -7236.324} C_VEL
LIN {X 0,Y 474.627,Z 398.865,A -85,B 0,C 180,E1 -7239.648,E2 -7239.648} C_VEL
LIN {X 0,Y 474.626,Z 398.865,A -85,B 0,C 180,E1 -7242.238,E2 -7242.238} C_VEL
LIN {X 0,Y 474.644,Z 399.154,A -85,B 0,C 180,E1 -7242.931,E2 -7242.931} C_VEL
LIN {X 0,Y 475.218,Z 402.808,A -85,B 0,C 180,E1 -7245.967,E2 -7245.967} C_VEL
LIN {X 0,Y 475.537,Z 405.898,A -85,B 0,C 180,E1 -7248.314,E2 -7248.314} C_VEL
LIN {X 0,Y 475.469,Z 409.059,A -85,B 0,C 180,E1 -7250.537,E2 -7250.537} C_VEL
LIN {X 0,Y 475.198,Z 412.806,A -85,B 0,C 180,E1 -7253.001,E2 -7253.001} C_VEL
LIN {X 0,Y 474.936,Z 417.552,A -85,B 0,C 180,E1 -7255.964,E2 -7255.964} C_VEL
LIN {X 0,Y 474.681,Z 422.354,A -85,B 0,C 180,E1 -7258.789,E2 -7258.789} C_VEL
LIN {X 0,Y 474.486,Z 427.547,A -85,B 0,C 180,E1 -7261.707,E2 -7261.707} C_VEL
LIN {X 0,Y 474.347,Z 433.033,A -85,B 0,C 180,E1 -7264.661,E2 -7264.661} C_VEL
LIN {X 0,Y 474.177,Z 438.164,A -85,B 0,C 180,E1 -7267.334,E2 -7267.334} C_VEL
LIN {X 0,Y 474.189,Z 441.836,A -85,B 0,C 180,E1 -7269.163,E2 -7269.163} C_VEL
LIN {X 0,Y 473.992,Z 447.328,A -85,B 0,C 180,E1 -7271.858,E2 -7271.858} C_VEL
LIN {X 0,Y 473.974,Z 453.494,A -85,B 0,C 180,E1 -7274.852,E2 -7274.852} C_VEL
LIN {X 0,Y 476.035,Z 465.143,A -85,B 0,C 180,E1 -7275.23,E2 -7275.23} C_VEL
LIN {X 0,Y 476.999,Z 471.715,A -85,B 0,C 180,E1 -7275.494,E2 -7275.494} C_VEL
LIN {X 0,Y 476.712,Z 482.344,A -85,B 0,C 180,E1 -7275.976,E2 -7275.976} C_VEL
LIN {X 0,Y 476.306,Z 492.47,A -85,B 0,C 180,E1 -7276.562,E2 -7276.562} C_VEL
LIN {X 0,Y 475.93,Z 501.443,A -85,B 0,C 180,E1 -7277.203,E2 -7277.203} C_VEL
LIN {X 0,Y 475.589,Z 510.15,A -85,B 0,C 180,E1 -7277.952,E2 -7277.952} C_VEL
LIN {X 0,Y 475.211,Z 517.519,A -85,B 0,C 180,E1 -7278.699,E2 -7278.699} C_VEL
LIN {X 0,Y 474.889,Z 524.711,A -85,B 0,C 180,E1 -7279.555,E2 -7279.555} C_VEL
LIN {X 0,Y 474.606,Z 530.888,A -85,B 0,C 180,E1 -7280.41,E2 -7280.41} C_VEL
LIN {X 0,Y 474.316,Z 537.395,A -85,B 0,C 180,E1 -7281.479,E2 -7281.479} C_VEL
LIN {X 0,Y 474.102,Z 541.874,A -85,B 0,C 180,E1 -7282.333,E2 -7282.333} C_VEL
LIN {X 0,Y 473.975,Z 546.727,A -85,B 0,C 180,E1 -7283.447,E2 -7283.447} C_VEL
LIN {X 0,Y 473.845,Z 551.627,A -85,B 0,C 180,E1 -7284.894,E2 -7284.894} C_VEL
LIN {X 0,Y 473.752,Z 553.973,A -85,B 0,C 180,E1 -7285.746,E2 -7285.746} C_VEL
LIN {X 0,Y 473.8,Z 555.76,A -85,B 0,C 180,E1 -7286.598,E2 -7286.598} C_VEL
LIN {X 0,Y 473.695,Z 558.186,A -85,B 0,C 180,E1 -7288.299,E2 -7288.299} C_VEL
LIN {X 0,Y 473.688,Z 558.769,A -85,B 0,C 180,E1 -7289.15,E2 -7289.15} C_VEL
LIN {X 0,Y 473.688,Z 558.769,A -85,B 0,C 180,E1 -7290.85,E2 -7290.85} C_VEL
LIN {X 0,Y 473.695,Z 558.186,A -85,B 0,C 180,E1 -7291.7,E2 -7291.7} C_VEL
LIN {X 0,Y 473.8,Z 555.761,A -85,B 0,C 180,E1 -7293.401,E2 -7293.401} C_VEL
LIN {X 0,Y 473.775,Z 552.836,A -85,B 0,C 180,E1 -7294.68,E2 -7294.68} C_VEL
LIN {X 0,Y 473.938,Z 548.878,A -85,B 0,C 180,E1 -7295.958,E2 -7295.958} C_VEL
LIN {X 0,Y 474.03,Z 543.78,A -85,B 0,C 180,E1 -7297.239,E2 -7297.239} C_VEL
LIN {X 0,Y 474.266,Z 538.547,A -85,B 0,C 180,E1 -7298.307,E2 -7298.307} C_VEL
LIN {X 0,Y 474.551,Z 532.26,A -85,B 0,C 180,E1 -7299.375,E2 -7299.375} C_VEL
LIN {X 0,Y 474.801,Z 526.335,A -85,B 0,C 180,E1 -7300.231,E2 -7300.231} C_VEL
LIN {X 0,Y 475.098,Z 519.435,A -85,B 0,C 180,E1 -7301.087,E2 -7301.087} C_VEL
LIN {X 0,Y 475.519,Z 511.283,A -85,B 0,C 180,E1 -7301.941,E2 -7301.941} C_VEL
LIN {X 0,Y 475.851,Z 504.147,A -85,B 0,C 180,E1 -7302.582,E2 -7302.582} C_VEL
LIN {X 0,Y 476.195,Z 494.59,A -85,B 0,C 180,E1 -7303.3,E2 -7303.3} C_VEL
LIN {X 0,Y 476.584,Z 484.362,A -85,B 0,C 180,E1 -7303.919,E2 -7303.919} C_VEL
LIN {X 0,Y 476.947,Z 474.297,A -85,B 0,C 180,E1 -7304.398,E2 -7304.398} C_VEL
LIN {X 0,Y 476.719,Z 469.078,A -85,B 0,C 180,E1 -7304.623,E2 -7304.623} C_VEL
LIN {X 0,Y 474.402,Z 456.03,A -85,B 0,C 180,E1 -7305.075,E2 -7305.075} C_VEL
LIN {X 0,Y 473.993,Z 453.492,A -85,B 0,C 180,E1 -7305.149,E2 -7305.149} C_VEL
LIN {X 0,Y 474.031,Z 445.5,A -85,B 0,C 180,E1 -7309.036,E2 -7309.036} C_VEL
LIN {X 0,Y 474.164,Z 440.002,A -85,B 0,C 180,E1 -7311.749,E2 -7311.749} C_VEL
LIN {X 0,Y 474.279,Z 434.605,A -85,B 0,C 180,E1 -7314.513,E2 -7314.513} C_VEL
LIN {X 0,Y 474.459,Z 429.292,A -85,B 0,C 180,E1 -7317.334,E2 -7317.334} C_VEL
LIN {X 0,Y 474.665,Z 423.014,A -85,B 0,C 180,E1 -7320.821,E2 -7320.821} C_VEL
LIN {X 0,Y 474.857,Z 418.924,A -85,B 0,C 180,E1 -7323.202,E2 -7323.202} C_VEL
LIN {X 0,Y 475.115,Z 413.91,A -85,B 0,C 180,E1 -7326.276,E2 -7326.276} C_VEL
LIN {X 0,Y 475.37,Z 410.616,A -85,B 0,C 180,E1 -7328.411,E2 -7328.411} C_VEL
LIN {X 0,Y 475.551,Z 406.708,A -85,B 0,C 180,E1 -7331.087,E2 -7331.087} C_VEL
LIN {X 0,Y 475.297,Z 403.398,A -85,B 0,C 180,E1 -7333.569,E2 -7333.569} C_VEL
LIN {X 0,Y 474.754,Z 399.833,A -85,B 0,C 180,E1 -7336.498,E2 -7336.498} C_VEL
LIN {X 0,Y 474.642,Z 399.166,A -85,B 0,C 180,E1 -7337.068,E2 -7337.068} C_VEL
LIN {X 0,Y 474.619,Z 398.866,A -85,B 0,C 180,E1 -7338.214,E2 -7338.214} C_VEL
LIN {X 0,Y 474.642,Z 398.863,A -85,B 0,C 180,E1 -7340.453,E2 -7340.453} C_VEL
LIN {X 0,Y 474.59,Z 398.868,A -85,B 0,C 180,E1 -7343.676,E2 -7343.676} C_VEL
LIN {X 0,Y 474.64,Z 398.864,A -85,B 0,C 180,E1 -7346.779,E2 -7346.779} C_VEL
LIN {X 0,Y 474.613,Z 398.86,A -85,B 0,C 180,E1 -7349.77,E2 -7349.77} C_VEL
LIN {X 0,Y 474.693,Z 398.857,A -85,B 0,C 180,E1 -7352.679,E2 -7352.679} C_VEL
LIN {X 0,Y 474.654,Z 398.856,A -85,B 0,C 180,E1 -7355.506,E2 -7355.506} C_VEL
LIN {X 0,Y 474.665,Z 398.856,A -85,B 0,C 180,E1 -7359.185,E2 -7359.185} C_VEL
LIN {X 0,Y 474.652,Z 398.856,A -85,B 0,C 180,E1 -7361.884,E2 -7361.884} C_VEL
LIN {X 0,Y 474.694,Z 398.858,A -85,B 0,C 180,E1 -7364.544,E2 -7364.544} C_VEL
LIN {X 0,Y 474.698,Z 398.852,A -85,B 0,C 180,E1 -7368.037,E2 -7368.037} C_VEL
LIN {X 0,Y 474.722,Z 398.847,A -85,B 0,C 180,E1 -7371.486,E2 -7371.486} C_VEL
LIN {X 0,Y 474.773,Z 398.843,A -85,B 0,C 180,E1 -7374.052,E2 -7374.052} C_VEL
LIN {X 0,Y 474.889,Z 398.826,A -85,B 0,C 180,E1 -7377.455,E2 -7377.455} C_VEL
LIN {X 0,Y 474.905,Z 398.827,A -85,B 0,C 180,E1 -7380,E2 -7380} C_VEL
LIN {X 0,Y 474.888,Z 398.832,A -85,B 0,C 180,E1 -7382.544,E2 -7382.544} C_VEL
LIN {X 0,Y 474.773,Z 398.844,A -85,B 0,C 180,E1 -7385.947,E2 -7385.947} C_VEL
LIN {X 0,Y 474.721,Z 398.852,A -85,B 0,C 180,E1 -7388.513,E2 -7388.513} C_VEL
LIN {X 0,Y 474.696,Z 398.855,A -85,B 0,C 180,E1 -7391.962,E2 -7391.962} C_VEL
LIN {X 0,Y 474.694,Z 398.854,A -85,B 0,C 180,E1 -7395.777,E2 -7395.777} C_VEL
LIN {X 0,Y 474.657,Z 398.855,A -85,B 0,C 180,E1 -7399.01,E2 -7399.01} C_VEL
LIN {X 0,Y 474.583,Z 398.868,A -85,B 0,C 180,E1 -7401.729,E2 -7401.729} C_VEL
LIN {X 0,Y 474.652,Z 398.858,A -85,B 0,C 180,E1 -7404.493,E2 -7404.493} C_VEL
LIN {X 0,Y 474.691,Z 398.852,A -85,B 0,C 180,E1 -7407.339,E2 -7407.339} C_VEL
LIN {X 0,Y 474.602,Z 398.862,A -85,B 0,C 180,E1 -7410.811,E2 -7410.811} C_VEL
LIN {X 0,Y 474.631,Z 398.865,A -85,B 0,C 180,E1 -7413.984,E2 -7413.984} C_VEL
LIN {X 0,Y 474.568,Z 398.866,A -85,B 0,C 180,E1 -7416.9,E2 -7416.9} C_VEL
LIN {X 0,Y 474.648,Z 398.863,A -85,B 0,C 180,E1 -7419.652,E2 -7419.652} C_VEL
LIN {X 0,Y 474.645,Z 398.857,A -85,B 0,C 180,E1 -7422.93,E2 -7422.93} C_VEL
LIN {X 0,Y 474.611,Z 398.866,A -85,B 0,C 180,E1 -7425.896,E2 -7425.896} C_VEL
LIN {X 0,Y 474.639,Z 398.859,A -85,B 0,C 180,E1 -7429.038,E2 -7429.038} C_VEL
LIN {X 0,Y 474.61,Z 398.868,A -85,B 0,C 180,E1 -7431.703,E2 -7431.703} C_VEL
LIN {X 0,Y 474.624,Z 398.859,A -85,B 0,C 180,E1 -7434.726,E2 -7434.726} C_VEL
LIN {X 0,Y 474.632,Z 398.862,A -85,B 0,C 180,E1 -7437.788,E2 -7437.788} C_VEL
LIN {X 0,Y 474.619,Z 398.861,A -85,B 0,C 180,E1 -7440.885,E2 -7440.885} C_VEL
LIN {X 0,Y 474.662,Z 398.86,A -85,B 0,C 180,E1 -7443.629,E2 -7443.629} C_VEL
LIN {X 0,Y 474.63,Z 398.859,A -85,B 0,C 180,E1 -7446.642,E2 -7446.642} C_VEL
LIN {X 0,Y 474.652,Z 398.856,A -85,B 0,C 180,E1 -7450.09,E2 -7450.09} C_VEL
LIN {X 0,Y 474.651,Z 398.861,A -85,B 0,C 180,E1 -7451.677,E2 -7451.677} C_VEL
LIN {X 0,Y 473.988,Z 398.941,A -85,B 0,C 180,E1 -7452.386,E2 -7452.386} C_VEL
LIN {X 0,Y 471.138,Z 399.301,A -85,B 0,C 180,E1 -7453.538,E2 -7453.538} C_VEL
LIN {X 0,Y 468.721,Z 399.604,A -85,B 0,C 180,E1 -7454.466,E2 -7454.466} C_VEL
LIN {X 0,Y 467.68,Z 399.732,A -85,B 0,C 180,E1 -7455.183,E2 -7455.183} C_VEL
LIN {X 0,Y 467.593,Z 399.741,A -85,B 0,C 180,E1 -7455.426,E2 -7455.426} C_VEL
LIN {X 0,Y 467.65,Z 399.732,A -85,B 0,C 180,E1 -7458.734,E2 -7458.734} C_VEL
LIN {X 0,Y 467.745,Z 399.719,A -85,B 0,C 180,E1 -7462.229,E2 -7462.229} C_VEL
LIN {X 0,Y 467.723,Z 399.725,A -85,B 0,C 180,E1 -7464.828,E2 -7464.828} C_VEL
LIN {X 0,Y 467.857,Z 399.708,A -85,B 0,C 180,E1 -7467.417,E2 -7467.417} C_VEL
LIN {X 0,Y 467.88,Z 399.703,A -85,B 0,C 180,E1 -7470,E2 -7470} C_VEL
LIN {X 0,Y 467.857,Z 399.708,A -85,B 0,C 180,E1 -7472.583,E2 -7472.583} C_VEL
LIN {X 0,Y 467.743,Z 399.72,A -85,B 0,C 180,E1 -7476.037,E2 -7476.037} C_VEL
LIN {X 0,Y 467.679,Z 399.731,A -85,B 0,C 180,E1 -7478.643,E2 -7478.643} C_VEL
LIN {X 0,Y 467.652,Z 399.73,A -85,B 0,C 180,E1 -7482.146,E2 -7482.146} C_VEL
LIN {X 0,Y 467.635,Z 399.733,A -85,B 0,C 180,E1 -7485.695,E2 -7485.695} C_VEL
LIN {X 0,Y 467.614,Z 399.741,A -85,B 0,C 180,E1 -7488.765,E2 -7488.765} C_VEL
LIN {X 0,Y 467.577,Z 399.738,A -85,B 0,C 180,E1 -7491.269,E2 -7491.269} C_VEL
LIN {X 0,Y 467.569,Z 399.739,A -85,B 0,C 180,E1 -7493.943,E2 -7493.943} C_VEL
LIN {X 0,Y 467.624,Z 399.736,A -85,B 0,C 180,E1 -7496.8,E2 -7496.8} C_VEL
LIN {X 0,Y 467.55,Z 399.741,A -85,B 0,C 180,E1 -7499.738,E2 -7499.738} C_VEL
LIN {X 0,Y 467.579,Z 399.741,A -85,B 0,C 180,E1 -7502.758,E2 -7502.758} C_VEL
LIN {X 0,Y 467.552,Z 399.742,A -85,B 0,C 180,E1 -7505.889,E2 -7505.889} C_VEL
LIN {X 0,Y 467.595,Z 399.735,A -85,B 0,C 180,E1 -7509.143,E2 -7509.143} C_VEL
LIN {X 0,Y 467.614,Z 399.737,A -85,B 0,C 180,E1 -7512.571,E2 -7512.571} C_VEL
LIN {X 0,Y 467.565,Z 399.739,A -85,B 0,C 180,E1 -7515.053,E2 -7515.053} C_VEL
LIN {X 0,Y 467.583,Z 399.736,A -85,B 0,C 180,E1 -7517.44,E2 -7517.44} C_VEL
LIN {X 0,Y 467.577,Z 399.738,A -85,B 0,C 180,E1 -7520.856,E2 -7520.856} C_VEL
LIN {X 0,Y 467.558,Z 399.746,A -85,B 0,C 180,E1 -7524.26,E2 -7524.26} C_VEL
LIN {X 0,Y 467.577,Z 399.737,A -85,B 0,C 180,E1 -7527.321,E2 -7527.321} C_VEL
LIN {X 0,Y 467.573,Z 399.739,A -85,B 0,C 180,E1 -7530.666,E2 -7530.666} C_VEL
LIN {X 0,Y 467.611,Z 399.733,A -85,B 0,C 180,E1 -7533.2,E2 -7533.2} C_VEL
LIN {X 0,Y 467.588,Z 399.738,A -85,B 0,C 180,E1 -7536.468,E2 -7536.468} C_VEL
LIN {X 0,Y 467.618,Z 399.738,A -85,B 0,C 180,E1 -7539.778,E2 -7539.778} C_VEL
LIN {X 0,Y 467.604,Z 399.735,A -85,B 0,C 180,E1 -7542.507,E2 -7542.507} C_VEL
LIN {X 0,Y 467.602,Z 399.735,A -85,B 0,C 180,E1 -7545.197,E2 -7545.197} C_VEL
LIN {X 0,Y 467.651,Z 399.735,A -85,B 0,C 180,E1 -7547.855,E2 -7547.855} C_VEL
LIN {X 0,Y 467.678,Z 399.728,A -85,B 0,C 180,E1 -7551.358,E2 -7551.358} C_VEL
LIN {X 0,Y 467.739,Z 399.721,A -85,B 0,C 180,E1 -7553.963,E2 -7553.963} C_VEL
LIN {X 0,Y 467.856,Z 399.707,A -85,B 0,C 180,E1 -7557.418,E2 -7557.418} C_VEL
LIN {X 0,Y 467.878,Z 399.703,A -85,B 0,C 180,E1 -7560,E2 -7560} C_VEL
LIN {X 0,Y 467.856,Z 399.702,A -85,B 0,C 180,E1 -7562.583,E2 -7562.583} C_VEL
LIN {X 0,Y 467.74,Z 399.719,A -85,B 0,C 180,E1 -7566.038,E2 -7566.038} C_VEL
LIN {X 0,Y 467.678,Z 399.724,A -85,B 0,C 180,E1 -7568.643,E2 -7568.643} C_VEL
LIN {X 0,Y 467.652,Z 399.728,A -85,B 0,C 180,E1 -7572.146,E2 -7572.146} C_VEL
LIN {X 0,Y 467.636,Z 399.733,A -85,B 0,C 180,E1 -7575.696,E2 -7575.696} C_VEL
LIN {X 0,Y 467.615,Z 399.734,A -85,B 0,C 180,E1 -7578.765,E2 -7578.765} C_VEL
LIN {X 0,Y 467.578,Z 399.745,A -85,B 0,C 180,E1 -7581.269,E2 -7581.269} C_VEL
LIN {X 0,Y 467.571,Z 399.738,A -85,B 0,C 180,E1 -7583.944,E2 -7583.944} C_VEL
LIN {X 0,Y 467.614,Z 399.735,A -85,B 0,C 180,E1 -7586.801,E2 -7586.801} C_VEL
LIN {X 0,Y 467.553,Z 399.741,A -85,B 0,C 180,E1 -7589.739,E2 -7589.739} C_VEL
LIN {X 0,Y 467.583,Z 399.74,A -85,B 0,C 180,E1 -7592.759,E2 -7592.759} C_VEL
LIN {X 0,Y 467.556,Z 399.742,A -85,B 0,C 180,E1 -7595.89,E2 -7595.89} C_VEL
LIN {X 0,Y 467.582,Z 399.745,A -85,B 0,C 180,E1 -7599.145,E2 -7599.145} C_VEL
LIN {X 0,Y 467.577,Z 399.744,A -85,B 0,C 180,E1 -7601.403,E2 -7601.403} C_VEL
LIN {X 0,Y 467.619,Z 399.994,A -85,B 0,C 180,E1 -7602.572,E2 -7602.572} C_VEL
LIN {X 0,Y 468.258,Z 404.16,A -85,B 0,C 180,E1 -7606.09,E2 -7606.09} C_VEL
LIN {X 0,Y 468.537,Z 407.567,A -85,B 0,C 180,E1 -7608.701,E2 -7608.701} C_VEL
LIN {X 0,Y 468.39,Z 411.251,A -85,B 0,C 180,E1 -7611.283,E2 -7611.283} C_VEL
LIN {X 0,Y 468.066,Z 415.657,A -85,B 0,C 180,E1 -7614.176,E2 -7614.176} C_VEL
LIN {X 0,Y 467.782,Z 420.697,A -85,B 0,C 180,E1 -7617.283,E2 -7617.283} C_VEL
LIN {X 0,Y 467.527,Z 425.773,A -85,B 0,C 180,E1 -7620.26,E2 -7620.26} C_VEL
LIN {X 0,Y 467.353,Z 431.008,A -85,B 0,C 180,E1 -7623.184,E2 -7623.184} C_VEL
LIN {X 0,Y 467.174,Z 436.314,A -85,B 0,C 180,E1 -7626.035,E2 -7626.035} C_VEL
LIN {X 0,Y 467.116,Z 441.823,A -85,B 0,C 180,E1 -7628.88,E2 -7628.88} C_VEL
LIN {X 0,Y 466.858,Z 449.042,A -85,B 0,C 180,E1 -7632.478,E2 -7632.478} C_VEL
LIN {X 0,Y 466.875,Z 453.357,A -85,B 0,C 180,E1 -7634.618,E2 -7634.618} C_VEL
LIN {X 0,Y 469.04,Z 465.21,A -85,B 0,C 180,E1 -7635.013,E2 -7635.013} C_VEL
LIN {X 0,Y 470.09,Z 472.847,A -85,B 0,C 180,E1 -7635.332,E2 -7635.332} C_VEL
LIN {X 0,Y 469.821,Z 482.208,A -85,B 0,C 180,E1 -7635.766,E2 -7635.766} C_VEL
LIN {X 0,Y 469.394,Z 492.357,A -85,B 0,C 180,E1 -7636.36,E2 -7636.36} C_VEL
LIN {X 0,Y 468.982,Z 501.355,A -85,B 0,C 180,E1 -7637.01,E2 -7637.01} C_VEL
LIN {X 0,Y 468.633,Z 510.166,A -85,B 0,C 180,E1 -7637.778,E2 -7637.778} C_VEL
LIN {X 0,Y 468.235,Z 517.488,A -85,B 0,C 180,E1 -7638.529,E2 -7638.529} C_VEL
LIN {X 0,Y 467.886,Z 524.707,A -85,B 0,C 180,E1 -7639.397,E2 -7639.397} C_VEL
LIN {X 0,Y 467.584,Z 530.883,A -85,B 0,C 180,E1 -7640.265,E2 -7640.265} C_VEL
LIN {X 0,Y 467.287,Z 537.391,A -85,B 0,C 180,E1 -7641.35,E2 -7641.35} C_VEL
LIN {X 0,Y 467.046,Z 541.869,A -85,B 0,C 180,E1 -7642.216,E2 -7642.216} C_VEL
LIN {X 0,Y 466.868,Z 547.205,A -85,B 0,C 180,E1 -7643.483,E2 -7643.483} C_VEL
LIN {X 0,Y 466.783,Z 551.624,A -85,B 0,C 180,E1 -7644.817,E2 -7644.817} C_VEL
LIN {X 0,Y 466.663,Z 553.972,A -85,B 0,C 180,E1 -7645.681,E2 -7645.681} C_VEL
LIN {X 0,Y 466.695,Z 555.757,A -85,B 0,C 180,E1 -7646.546,E2 -7646.546} C_VEL
LIN {X 0,Y 466.604,Z 558.182,A -85,B 0,C 180,E1 -7648.274,E2 -7648.274} C_VEL
LIN {X 0,Y 466.59,Z 558.765,A -85,B 0,C 180,E1 -7649.137,E2 -7649.137} C_VEL
LIN {X 0,Y 466.59,Z 558.766,A -85,B 0,C 180,E1 -7650.863,E2 -7650.863} C_VEL
LIN {X 0,Y 466.604,Z 558.182,A -85,B 0,C 180,E1 -7651.726,E2 -7651.726} C_VEL
LIN {X 0,Y 466.695,Z 555.758,A -85,B 0,C 180,E1 -7653.453,E2 -7653.453} C_VEL
LIN {X 0,Y 466.703,Z 552.833,A -85,B 0,C 180,E1 -7654.751,E2 -7654.751} C_VEL
LIN {X 0,Y 466.836,Z 548.874,A -85,B 0,C 180,E1 -7656.049,E2 -7656.049} C_VEL
LIN {X 0,Y 466.96,Z 543.776,A -85,B 0,C 180,E1 -7657.35,E2 -7657.35} C_VEL
LIN {X 0,Y 467.207,Z 538.543,A -85,B 0,C 180,E1 -7658.433,E2 -7658.433} C_VEL
LIN {X 0,Y 467.508,Z 532.256,A -85,B 0,C 180,E1 -7659.518,E2 -7659.518} C_VEL
LIN {X 0,Y 467.784,Z 526.33,A -85,B 0,C 180,E1 -7660.386,E2 -7660.386} C_VEL
LIN {X 0,Y 468.125,Z 519.411,A -85,B 0,C 180,E1 -7661.254,E2 -7661.254} C_VEL
LIN {X 0,Y 468.557,Z 511.229,A -85,B 0,C 180,E1 -7662.121,E2 -7662.121} C_VEL
LIN {X 0,Y 468.935,Z 502.897,A -85,B 0,C 180,E1 -7662.866,E2 -7662.866} C_VEL
LIN {X 0,Y 469.328,Z 493.997,A -85,B 0,C 180,E1 -7663.531,E2 -7663.531} C_VEL
LIN {X 0,Y 469.708,Z 484.229,A -85,B 0,C 180,E1 -7664.127,E2 -7664.127} C_VEL
LIN {X 0,Y 470.054,Z 474.144,A -85,B 0,C 180,E1 -7664.614,E2 -7664.614} C_VEL
LIN {X 0,Y 469.571,Z 468.709,A -85,B 0,C 180,E1 -7664.858,E2 -7664.858} C_VEL
LIN {X 0,Y 467.333,Z 455.867,A -85,B 0,C 180,E1 -7665.307,E2 -7665.307} C_VEL
LIN {X 0,Y 466.904,Z 453.327,A -85,B 0,C 180,E1 -7665.396,E2 -7665.396} C_VEL
LIN {X 0,Y 466.941,Z 447.039,A -85,B 0,C 180,E1 -7668.517,E2 -7668.517} C_VEL
LIN {X 0,Y 467.099,Z 441.73,A -85,B 0,C 180,E1 -7671.168,E2 -7671.168} C_VEL
LIN {X 0,Y 467.172,Z 436.306,A -85,B 0,C 180,E1 -7673.964,E2 -7673.964} C_VEL
LIN {X 0,Y 467.345,Z 430.99,A -85,B 0,C 180,E1 -7676.816,E2 -7676.816} C_VEL
LIN {X 0,Y 467.52,Z 425.759,A -85,B 0,C 180,E1 -7679.74,E2 -7679.74} C_VEL
LIN {X 0,Y 467.781,Z 420.635,A -85,B 0,C 180,E1 -7682.742,E2 -7682.742} C_VEL
LIN {X 0,Y 468.065,Z 415.61,A -85,B 0,C 180,E1 -7685.843,E2 -7685.843} C_VEL
LIN {X 0,Y 468.4,Z 410.728,A -85,B 0,C 180,E1 -7689.062,E2 -7689.062} C_VEL
LIN {X 0,Y 468.549,Z 407.406,A -85,B 0,C 180,E1 -7691.411,E2 -7691.411} C_VEL
LIN {X 0,Y 468.256,Z 404.161,A -85,B 0,C 180,E1 -7693.91,E2 -7693.91} C_VEL
LIN {X 0,Y 467.617,Z 399.996,A -85,B 0,C 180,E1 -7697.428,E2 -7697.428} C_VEL
LIN {X 0,Y 467.58,Z 399.742,A -85,B 0,C 180,E1 -7700.045,E2 -7700.045} C_VEL
LIN {X 0,Y 467.53,Z 399.751,A -85,B 0,C 180,E1 -7703.037,E2 -7703.037} C_VEL
LIN {X 0,Y 467.583,Z 399.737,A -85,B 0,C 180,E1 -7706.211,E2 -7706.211} C_VEL
LIN {X 0,Y 467.578,Z 399.74,A -85,B 0,C 180,E1 -7709.266,E2 -7709.266} C_VEL
LIN {X 0,Y 467.641,Z 399.732,A -85,B 0,C 180,E1 -7712.458,E2 -7712.458} C_VEL
LIN {X 0,Y 467.599,Z 399.738,A -85,B 0,C 180,E1 -7715.112,E2 -7715.112} C_VEL
LIN {X 0,Y 467.529,Z 399.743,A -85,B 0,C 180,E1 -7717.925,E2 -7717.925} C_VEL
LIN {X 0,Y 467.618,Z 399.74,A -85,B 0,C 180,E1 -7720.692,E2 -7720.692} C_VEL
LIN {X 0,Y 467.644,Z 399.73,A -85,B 0,C 180,E1 -7724.114,E2 -7724.114} C_VEL
LIN {X 0,Y 467.647,Z 399.728,A -85,B 0,C 180,E1 -7727.642,E2 -7727.642} C_VEL
LIN {X 0,Y 467.659,Z 399.734,A -85,B 0,C 180,E1 -7730.484,E2 -7730.484} C_VEL
LIN {X 0,Y 467.705,Z 399.722,A -85,B 0,C 180,E1 -7733.095,E2 -7733.095} C_VEL
LIN {X 0,Y 467.719,Z 399.723,A -85,B 0,C 180,E1 -7734.827,E2 -7734.827} C_VEL
LIN {X 0,Y 467.854,Z 399.702,A -85,B 0,C 180,E1 -7737.417,E2 -7737.417} C_VEL
LIN {X 0,Y 467.876,Z 399.703,A -85,B 0,C 180,E1 -7740,E2 -7740} C_VEL
LIN {X 0,Y 467.854,Z 399.707,A -85,B 0,C 180,E1 -7742.582,E2 -7742.582} C_VEL
LIN {X 0,Y 467.737,Z 399.722,A -85,B 0,C 180,E1 -7746.037,E2 -7746.037} C_VEL
LIN {X 0,Y 467.675,Z 399.728,A -85,B 0,C 180,E1 -7748.642,E2 -7748.642} C_VEL
LIN {X 0,Y 467.648,Z 399.736,A -85,B 0,C 180,E1 -7752.145,E2 -7752.145} C_VEL
LIN {X 0,Y 467.659,Z 399.731,A -85,B 0,C 180,E1 -7755.893,E2 -7755.893} C_VEL
LIN {X 0,Y 467.615,Z 399.732,A -85,B 0,C 180,E1 -7759.308,E2 -7759.308} C_VEL
LIN {X 0,Y 467.529,Z 399.751,A -85,B 0,C 180,E1 -7762.074,E2 -7762.074} C_VEL
LIN {X 0,Y 467.596,Z 399.735,A -85,B 0,C 180,E1 -7764.887,E2 -7764.887} C_VEL
LIN {X 0,Y 467.621,Z 399.737,A -85,B 0,C 180,E1 -7767.768,E2 -7767.768} C_VEL
LIN {X 0,Y 467.565,Z 399.739,A -85,B 0,C 180,E1 -7771.046,E2 -7771.046} C_VEL
LIN {X 0,Y 467.583,Z 399.739,A -85,B 0,C 180,E1 -7774.243,E2 -7774.243} C_VEL
LIN {X 0,Y 467.545,Z 399.742,A -85,B 0,C 180,E1 -7777.187,E2 -7777.187} C_VEL
LIN {X 0,Y 467.59,Z 399.737,A -85,B 0,C 180,E1 -7780.263,E2 -7780.263} C_VEL
LIN {X 0,Y 467.612,Z 399.733,A -85,B 0,C 180,E1 -7782.571,E2 -7782.571} C_VEL
LIN {X 0,Y 467.567,Z 399.74,A -85,B 0,C 180,E1 -7786.177,E2 -7786.177} C_VEL
LIN {X 0,Y 467.583,Z 399.736,A -85,B 0,C 180,E1 -7788.722,E2 -7788.722} C_VEL
LIN {X 0,Y 467.564,Z 399.742,A -85,B 0,C 180,E1 -7791.956,E2 -7791.956} C_VEL
LIN {X 0,Y 467.563,Z 399.742,A -85,B 0,C 180,E1 -7795.168,E2 -7795.168} C_VEL
LIN {X 0,Y 467.578,Z 399.737,A -85,B 0,C 180,E1 -7798.26,E2 -7798.26} C_VEL
LIN {X 0,Y 467.572,Z 399.743,A -85,B 0,C 180,E1 -7801.251,E2 -7801.251} C_VEL
LIN {X 0,Y 467.607,Z 399.734,A -85,B 0,C 180,E1 -7804.16,E2 -7804.16} C_VEL
LIN {X 0,Y 467.572,Z 399.741,A -85,B 0,C 180,E1 -7806.996,E2 -7806.996} C_VEL
LIN {X 0,Y 467.619,Z 399.736,A -85,B 0,C 180,E1 -7809.778,E2 -7809.778} C_VEL
LIN {X 0,Y 467.604,Z 399.737,A -85,B 0,C 180,E1 -7812.507,E2 -7812.507} C_VEL
LIN {X 0,Y 467.593,Z 399.741,A -85,B 0,C 180,E1 -7815.426,E2 -7815.426} C_VEL
LIN {X 0,Y 466.922,Z 399.822,A -85,B 0,C 180,E1 -7816.146,E2 -7816.146} C_VEL
LIN {X 0,Y 464.079,Z 400.18,A -85,B 0,C 180,E1 -7817.314,E2 -7817.314} C_VEL
LIN {X 0,Y 461.681,Z 400.475,A -85,B 0,C 180,E1 -7818.256,E2 -7818.256} C_VEL
LIN {X 0,Y 460.656,Z 400.607,A -85,B 0,C 180,E1 -7818.984,E2 -7818.984} C_VEL
LIN {X 0,Y 460.574,Z 400.614,A -85,B 0,C 180,E1 -7819.23,E2 -7819.23} C_VEL
LIN {X 0,Y 460.716,Z 400.597,A -85,B 0,C 180,E1 -7822.539,E2 -7822.539} C_VEL
LIN {X 0,Y 460.696,Z 400.6,A -85,B 0,C 180,E1 -7824.749,E2 -7824.749} C_VEL
LIN {X 0,Y 460.822,Z 400.585,A -85,B 0,C 180,E1 -7827.378,E2 -7827.378} C_VEL
LIN {X 0,Y 460.85,Z 400.579,A -85,B 0,C 180,E1 -7830,E2 -7830} C_VEL
LIN {X 0,Y 460.822,Z 400.585,A -85,B 0,C 180,E1 -7832.623,E2 -7832.623} C_VEL
LIN {X 0,Y 460.709,Z 400.597,A -85,B 0,C 180,E1 -7836.13,E2 -7836.13} C_VEL
LIN {X 0,Y 460.626,Z 400.611,A -85,B 0,C 180,E1 -7838.776,E2 -7838.776} C_VEL
LIN {X 0,Y 460.61,Z 400.609,A -85,B 0,C 180,E1 -7842.445,E2 -7842.445} C_VEL
LIN {X 0,Y 460.596,Z 400.61,A -85,B 0,C 180,E1 -7845.998,E2 -7845.998} C_VEL
LIN {X 0,Y 460.568,Z 400.618,A -85,B 0,C 180,E1 -7848.902,E2 -7848.902} C_VEL
LIN {X 0,Y 460.512,Z 400.617,A -85,B 0,C 180,E1 -7851.486,E2 -7851.486} C_VEL
LIN {X 0,Y 460.539,Z 400.618,A -85,B 0,C 180,E1 -7854.332,E2 -7854.332} C_VEL
LIN {X 0,Y 460.58,Z 400.609,A -85,B 0,C 180,E1 -7857.243,E2 -7857.243} C_VEL
LIN {X 0,Y 460.507,Z 400.622,A -85,B 0,C 180,E1 -7860.24,E2 -7860.24} C_VEL
LIN {X 0,Y 460.525,Z 400.616,A -85,B 0,C 180,E1 -7863.325,E2 -7863.325} C_VEL
LIN {X 0,Y 460.475,Z 400.629,A -85,B 0,C 180,E1 -7866.529,E2 -7866.529} C_VEL
LIN {X 0,Y 460.57,Z 400.612,A -85,B 0,C 180,E1 -7869.858,E2 -7869.858} C_VEL
LIN {X 0,Y 460.537,Z 400.615,A -85,B 0,C 180,E1 -7872.904,E2 -7872.904} C_VEL
LIN {X 0,Y 460.506,Z 400.62,A -85,B 0,C 180,E1 -7875.83,E2 -7875.83} C_VEL
LIN {X 0,Y 460.526,Z 400.616,A -85,B 0,C 180,E1 -7878.989,E2 -7878.989} C_VEL
LIN {X 0,Y 460.521,Z 400.616,A -85,B 0,C 180,E1 -7881.267,E2 -7881.267} C_VEL
LIN {X 0,Y 460.508,Z 400.621,A -85,B 0,C 180,E1 -7884.555,E2 -7884.555} C_VEL
LIN {X 0,Y 460.528,Z 400.618,A -85,B 0,C 180,E1 -7887.716,E2 -7887.716} C_VEL
LIN {X 0,Y 460.542,Z 400.614,A -85,B 0,C 180,E1 -7890.77,E2 -7890.77} C_VEL
LIN {X 0,Y 460.558,Z 400.616,A -85,B 0,C 180,E1 -7893.735,E2 -7893.735} C_VEL
LIN {X 0,Y 460.541,Z 400.614,A -85,B 0,C 180,E1 -7896.624,E2 -7896.624} C_VEL
LIN {X 0,Y 460.546,Z 400.615,A -85,B 0,C 180,E1 -7899.453,E2 -7899.453} C_VEL
LIN {X 0,Y 460.555,Z 400.615,A -85,B 0,C 180,E1 -7902.231,E2 -7902.231} C_VEL
LIN {X 0,Y 460.565,Z 400.611,A -85,B 0,C 180,E1 -7904.965,E2 -7904.965} C_VEL
LIN {X 0,Y 460.607,Z 400.606,A -85,B 0,C 180,E1 -7908.56,E2 -7908.56} C_VEL
LIN {X 0,Y 460.691,Z 400.598,A -85,B 0,C 180,E1 -7912.109,E2 -7912.109} C_VEL
LIN {X 0,Y 460.694,Z 400.594,A -85,B 0,C 180,E1 -7914.749,E2 -7914.749} C_VEL
LIN {X 0,Y 460.821,Z 400.583,A -85,B 0,C 180,E1 -7917.378,E2 -7917.378} C_VEL
LIN {X 0,Y 460.849,Z 400.578,A -85,B 0,C 180,E1 -7920,E2 -7920} C_VEL
LIN {X 0,Y 460.821,Z 400.578,A -85,B 0,C 180,E1 -7922.623,E2 -7922.623} C_VEL
LIN {X 0,Y 460.706,Z 400.594,A -85,B 0,C 180,E1 -7926.13,E2 -7926.13} C_VEL
LIN {X 0,Y 460.626,Z 400.604,A -85,B 0,C 180,E1 -7928.777,E2 -7928.777} C_VEL
LIN {X 0,Y 460.61,Z 400.605,A -85,B 0,C 180,E1 -7932.445,E2 -7932.445} C_VEL
LIN {X 0,Y 460.597,Z 400.607,A -85,B 0,C 180,E1 -7935.998,E2 -7935.998} C_VEL
LIN {X 0,Y 460.568,Z 400.613,A -85,B 0,C 180,E1 -7938.902,E2 -7938.902} C_VEL
LIN {X 0,Y 460.513,Z 400.622,A -85,B 0,C 180,E1 -7941.486,E2 -7941.486} C_VEL
LIN {X 0,Y 460.54,Z 400.614,A -85,B 0,C 180,E1 -7944.333,E2 -7944.333} C_VEL
LIN {X 0,Y 460.572,Z 400.617,A -85,B 0,C 180,E1 -7947.244,E2 -7947.244} C_VEL
LIN {X 0,Y 460.51,Z 400.617,A -85,B 0,C 180,E1 -7950.241,E2 -7950.241} C_VEL
LIN {X 0,Y 460.528,Z 400.621,A -85,B 0,C 180,E1 -7953.325,E2 -7953.325} C_VEL
LIN {X 0,Y 460.478,Z 400.626,A -85,B 0,C 180,E1 -7956.53,E2 -7956.53} C_VEL
LIN {X 0,Y 460.545,Z 400.621,A -85,B 0,C 180,E1 -7958.898,E2 -7958.898} C_VEL
LIN {X 0,Y 460.533,Z 400.622,A -85,B 0,C 180,E1 -7961.603,E2 -7961.603} C_VEL
LIN {X 0,Y 460.527,Z 400.81,A -85,B 0,C 180,E1 -7962.181,E2 -7962.181} C_VEL
LIN {X 0,Y 461.145,Z 404.626,A -85,B 0,C 180,E1 -7965.489,E2 -7965.489} C_VEL
LIN {X 0,Y 461.508,Z 408.107,A -85,B 0,C 180,E1 -7968.262,E2 -7968.262} C_VEL
LIN {X 0,Y 461.381,Z 412.422,A -85,B 0,C 180,E1 -7971.353,E2 -7971.353} C_VEL
LIN {X 0,Y 460.983,Z 417.319,A -85,B 0,C 180,E1 -7974.597,E2 -7974.597} C_VEL
LIN {X 0,Y 460.703,Z 422.346,A -85,B 0,C 180,E1 -7977.729,E2 -7977.729} C_VEL
LIN {X 0,Y 460.436,Z 427.467,A -85,B 0,C 180,E1 -7980.762,E2 -7980.762} C_VEL
LIN {X 0,Y 460.267,Z 432.704,A -85,B 0,C 180,E1 -7983.717,E2 -7983.717} C_VEL
LIN {X 0,Y 460.073,Z 438.001,A -85,B 0,C 180,E1 -7986.599,E2 -7986.599} C_VEL
LIN {X 0,Y 459.976,Z 443.36,A -85,B 0,C 180,E1 -7989.426,E2 -7989.426} C_VEL
LIN {X 0,Y 459.788,Z 448.825,A -85,B 0,C 180,E1 -7992.199,E2 -7992.199} C_VEL
LIN {X 0,Y 459.74,Z 453.235,A -85,B 0,C 180,E1 -7994.382,E2 -7994.382} C_VEL
LIN {X 0,Y 461.714,Z 463.654,A -85,B 0,C 180,E1 -7994.727,E2 -7994.727} C_VEL
LIN {X 0,Y 463.079,Z 472.631,A -85,B 0,C 180,E1 -7995.105,E2 -7995.105} C_VEL
LIN {X 0,Y 462.942,Z 481.997,A -85,B 0,C 180,E1 -7995.55,E2 -7995.55} C_VEL
LIN {X 0,Y 462.45,Z 492.468,A -85,B 0,C 180,E1 -7996.174,E2 -7996.174} C_VEL
LIN {X 0,Y 462.022,Z 501.142,A -85,B 0,C 180,E1 -7996.811,E2 -7996.811} C_VEL
LIN {X 0,Y 461.722,Z 509.032,A -85,B 0,C 180,E1 -7997.501,E2 -7997.501} C_VEL
LIN {X 0,Y 461.257,Z 517.276,A -85,B 0,C 180,E1 -7998.353,E2 -7998.353} C_VEL
LIN {X 0,Y 460.868,Z 524.5,A -85,B 0,C 180,E1 -7999.234,E2 -7999.234} C_VEL
LIN {X 0,Y 460.556,Z 530.705,A -85,B 0,C 180,E1 -8000.115,E2 -8000.115} C_VEL
LIN {X 0,Y 460.236,Z 537.245,A -85,B 0,C 180,E1 -8001.216,E2 -8001.216} C_VEL
LIN {X 0,Y 459.983,Z 541.747,A -85,B 0,C 180,E1 -8002.096,E2 -8002.096} C_VEL
LIN {X 0,Y 459.783,Z 547.514,A -85,B 0,C 180,E1 -8003.495,E2 -8003.495} C_VEL
LIN {X 0,Y 459.699,Z 551.565,A -85,B 0,C 180,E1 -8004.737,E2 -8004.737} C_VEL
LIN {X 0,Y 459.58,Z 553.929,A -85,B 0,C 180,E1 -8005.615,E2 -8005.615} C_VEL
LIN {X 0,Y 459.591,Z 555.727,A -85,B 0,C 180,E1 -8006.493,E2 -8006.493} C_VEL
LIN {X 0,Y 459.517,Z 558.169,A -85,B 0,C 180,E1 -8008.247,E2 -8008.247} C_VEL
LIN {X 0,Y 459.495,Z 558.755,A -85,B 0,C 180,E1 -8009.123,E2 -8009.123} C_VEL
LIN {X 0,Y 459.495,Z 558.756,A -85,B 0,C 180,E1 -8010.876,E2 -8010.876} C_VEL
LIN {X 0,Y 459.517,Z 558.169,A -85,B 0,C 180,E1 -8011.753,E2 -8011.753} C_VEL
LIN {X 0,Y 459.591,Z 555.728,A -85,B 0,C 180,E1 -8013.507,E2 -8013.507} C_VEL
LIN {X 0,Y 459.634,Z 552.781,A -85,B 0,C 180,E1 -8014.824,E2 -8014.824} C_VEL
LIN {X 0,Y 459.754,Z 548.795,A -85,B 0,C 180,E1 -8016.142,E2 -8016.142} C_VEL
LIN {X 0,Y 459.884,Z 543.664,A -85,B 0,C 180,E1 -8017.463,E2 -8017.463} C_VEL
LIN {X 0,Y 460.174,Z 538.403,A -85,B 0,C 180,E1 -8018.563,E2 -8018.563} C_VEL
LIN {X 0,Y 460.479,Z 532.084,A -85,B 0,C 180,E1 -8019.665,E2 -8019.665} C_VEL
LIN {X 0,Y 460.762,Z 526.129,A -85,B 0,C 180,E1 -8020.546,E2 -8020.546} C_VEL
LIN {X 0,Y 461.125,Z 519.199,A -85,B 0,C 180,E1 -8021.427,E2 -8021.427} C_VEL
LIN {X 0,Y 461.588,Z 511.017,A -85,B 0,C 180,E1 -8022.307,E2 -8022.307} C_VEL
LIN {X 0,Y 461.952,Z 502.684,A -85,B 0,C 180,E1 -8023.064,E2 -8023.064} C_VEL
LIN {X 0,Y 462.407,Z 493.785,A -85,B 0,C 180,E1 -8023.737,E2 -8023.737} C_VEL
LIN {X 0,Y 462.752,Z 485.024,A -85,B 0,C 180,E1 -8024.288,E2 -8024.288} C_VEL
LIN {X 0,Y 463.16,Z 475.222,A -85,B 0,C 180,E1 -8024.78,E2 -8024.78} C_VEL
LIN {X 0,Y 462.723,Z 470.047,A -85,B 0,C 180,E1 -8025.019,E2 -8025.019} C_VEL
LIN {X 0,Y 460.332,Z 456.247,A -85,B 0,C 180,E1 -8025.533,E2 -8025.533} C_VEL
LIN {X 0,Y 459.779,Z 453.122,A -85,B 0,C 180,E1 -8025.635,E2 -8025.635} C_VEL
LIN {X 0,Y 459.857,Z 447.008,A -85,B 0,C 180,E1 -8028.719,E2 -8028.719} C_VEL
LIN {X 0,Y 460.014,Z 441.564,A -85,B 0,C 180,E1 -8031.51,E2 -8031.51} C_VEL
LIN {X 0,Y 460.139,Z 436.213,A -85,B 0,C 180,E1 -8034.354,E2 -8034.354} C_VEL
LIN {X 0,Y 460.349,Z 430.171,A -85,B 0,C 180,E1 -8037.69,E2 -8037.69} C_VEL
LIN {X 0,Y 460.519,Z 425.743,A -85,B 0,C 180,E1 -8040.239,E2 -8040.239} C_VEL
LIN {X 0,Y 460.763,Z 420.638,A -85,B 0,C 180,E1 -8043.305,E2 -8043.305} C_VEL
LIN {X 0,Y 461.081,Z 415.664,A -85,B 0,C 180,E1 -8046.473,E2 -8046.473} C_VEL
LIN {X 0,Y 461.381,Z 411.871,A -85,B 0,C 180,E1 -8049.026,E2 -8049.026} C_VEL
LIN {X 0,Y 461.504,Z 408.108,A -85,B 0,C 180,E1 -8051.738,E2 -8051.738} C_VEL
LIN {X 0,Y 461.147,Z 404.626,A -85,B 0,C 180,E1 -8054.51,E2 -8054.51} C_VEL
LIN {X 0,Y 460.524,Z 400.808,A -85,B 0,C 180,E1 -8057.818,E2 -8057.818} C_VEL
LIN {X 0,Y 460.53,Z 400.621,A -85,B 0,C 180,E1 -8060.137,E2 -8060.137} C_VEL
LIN {X 0,Y 460.524,Z 400.622,A -85,B 0,C 180,E1 -8062.518,E2 -8062.518} C_VEL
LIN {X 0,Y 460.545,Z 400.615,A -85,B 0,C 180,E1 -8065.623,E2 -8065.623} C_VEL
LIN {X 0,Y 460.533,Z 400.621,A -85,B 0,C 180,E1 -8068.744,E2 -8068.744} C_VEL
LIN {X 0,Y 460.554,Z 400.612,A -85,B 0,C 180,E1 -8071.767,E2 -8071.767} C_VEL
LIN {X 0,Y 460.554,Z 400.619,A -85,B 0,C 180,E1 -8074.705,E2 -8074.705} C_VEL
LIN {X 0,Y 460.506,Z 400.618,A -85,B 0,C 180,E1 -8077.571,E2 -8077.571} C_VEL
LIN {X 0,Y 460.564,Z 400.615,A -85,B 0,C 180,E1 -8080.384,E2 -8080.384} C_VEL
LIN {X 0,Y 460.56,Z 400.613,A -85,B 0,C 180,E1 -8083.146,E2 -8083.146} C_VEL
LIN {X 0,Y 460.552,Z 400.613,A -85,B 0,C 180,E1 -8085.867,E2 -8085.867} C_VEL
LIN {X 0,Y 460.605,Z 400.614,A -85,B 0,C 180,E1 -8088.559,E2 -8088.559} C_VEL
LIN {X 0,Y 460.689,Z 400.598,A -85,B 0,C 180,E1 -8092.108,E2 -8092.108} C_VEL
LIN {X 0,Y 460.692,Z 400.599,A -85,B 0,C 180,E1 -8094.748,E2 -8094.748} C_VEL
LIN {X 0,Y 460.819,Z 400.579,A -85,B 0,C 180,E1 -8097.377,E2 -8097.377} C_VEL
LIN {X 0,Y 460.846,Z 400.578,A -85,B 0,C 180,E1 -8100,E2 -8100} C_VEL
LIN {X 0,Y 460.819,Z 400.583,A -85,B 0,C 180,E1 -8102.622,E2 -8102.622} C_VEL
LIN {X 0,Y 460.703,Z 400.599,A -85,B 0,C 180,E1 -8106.129,E2 -8106.129} C_VEL
LIN {X 0,Y 460.622,Z 400.605,A -85,B 0,C 180,E1 -8108.776,E2 -8108.776} C_VEL
LIN {X 0,Y 460.606,Z 400.61,A -85,B 0,C 180,E1 -8112.445,E2 -8112.445} C_VEL
LIN {X 0,Y 460.614,Z 400.611,A -85,B 0,C 180,E1 -8116.007,E2 -8116.007} C_VEL
LIN {X 0,Y 460.561,Z 400.613,A -85,B 0,C 180,E1 -8119.615,E2 -8119.615} C_VEL
LIN {X 0,Y 460.505,Z 400.621,A -85,B 0,C 180,E1 -8122.428,E2 -8122.428} C_VEL
LIN {X 0,Y 460.561,Z 400.616,A -85,B 0,C 180,E1 -8125.802,E2 -8125.802} C_VEL
LIN {X 0,Y 460.551,Z 400.617,A -85,B 0,C 180,E1 -8128.232,E2 -8128.232} C_VEL
LIN {X 0,Y 460.517,Z 400.618,A -85,B 0,C 180,E1 -8131.284,E2 -8131.284} C_VEL
LIN {X 0,Y 460.527,Z 400.616,A -85,B 0,C 180,E1 -8134.506,E2 -8134.506} C_VEL
LIN {X 0,Y 460.524,Z 400.621,A -85,B 0,C 180,E1 -8137.62,E2 -8137.62} C_VEL
LIN {X 0,Y 460.553,Z 400.614,A -85,B 0,C 180,E1 -8140.272,E2 -8140.272} C_VEL
LIN {X 0,Y 460.518,Z 400.62,A -85,B 0,C 180,E1 -8143.372,E2 -8143.372} C_VEL
LIN {X 0,Y 460.518,Z 400.616,A -85,B 0,C 180,E1 -8146.628,E2 -8146.628} C_VEL
LIN {X 0,Y 460.552,Z 400.619,A -85,B 0,C 180,E1 -8149.728,E2 -8149.728} C_VEL
LIN {X 0,Y 460.522,Z 400.616,A -85,B 0,C 180,E1 -8152.519,E2 -8152.519} C_VEL
LIN {X 0,Y 460.543,Z 400.62,A -85,B 0,C 180,E1 -8155.624,E2 -8155.624} C_VEL
LIN {X 0,Y 460.531,Z 400.615,A -85,B 0,C 180,E1 -8158.745,E2 -8158.745} C_VEL
LIN {X 0,Y 460.583,Z 400.608,A -85,B 0,C 180,E1 -8162.252,E2 -8162.252} C_VEL
LIN {X 0,Y 460.554,Z 400.613,A -85,B 0,C 180,E1 -8164.706,E2 -8164.706} C_VEL
LIN {X 0,Y 460.507,Z 400.623,A -85,B 0,C 180,E1 -8167.572,E2 -8167.572} C_VEL
LIN {X 0,Y 460.565,Z 400.61,A -85,B 0,C 180,E1 -8170.385,E2 -8170.385} C_VEL
LIN {X 0,Y 460.561,Z 400.619,A -85,B 0,C 180,E1 -8173.146,E2 -8173.146} C_VEL
LIN {X 0,Y 460.551,Z 400.616,A -85,B 0,C 180,E1 -8175.868,E2 -8175.868} C_VEL
LIN {X 0,Y 460.608,Z 400.608,A -85,B 0,C 180,E1 -8178.56,E2 -8178.56} C_VEL
LIN {X 0,Y 460.574,Z 400.614,A -85,B 0,C 180,E1 -8179.23,E2 -8179.23} C_VEL
LIN {X 0,Y 459.92,Z 400.7,A -85,B 0,C 180,E1 -8179.96,E2 -8179.96} C_VEL
LIN {X 0,Y 457.101,Z 401.055,A -85,B 0,C 180,E1 -8181.147,E2 -8181.147} C_VEL
LIN {X 0,Y 454.722,Z 401.349,A -85,B 0,C 180,E1 -8182.104,E2 -8182.104} C_VEL
LIN {X 0,Y 453.71,Z 401.471,A -85,B 0,C 180,E1 -8182.843,E2 -8182.843} C_VEL
LIN {X 0,Y 453.633,Z 401.479,A -85,B 0,C 180,E1 -8183.093,E2 -8183.093} C_VEL
LIN {X 0,Y 453.669,Z 401.475,A -85,B 0,C 180,E1 -8184.667,E2 -8184.667} C_VEL
LIN {X 0,Y 453.762,Z 401.465,A -85,B 0,C 180,E1 -8187.337,E2 -8187.337} C_VEL
LIN {X 0,Y 453.821,Z 401.455,A -85,B 0,C 180,E1 -8190,E2 -8190} C_VEL
LIN {X 0,Y 453.762,Z 401.465,A -85,B 0,C 180,E1 -8192.663,E2 -8192.663} C_VEL
LIN {X 0,Y 453.676,Z 401.473,A -85,B 0,C 180,E1 -8196.225,E2 -8196.225} C_VEL
LIN {X 0,Y 453.589,Z 401.487,A -85,B 0,C 180,E1 -8198.913,E2 -8198.913} C_VEL
LIN {X 0,Y 453.56,Z 401.488,A -85,B 0,C 180,E1 -8202.529,E2 -8202.529} C_VEL
LIN {X 0,Y 453.541,Z 401.49,A -85,B 0,C 180,E1 -8206.196,E2 -8206.196} C_VEL
LIN {X 0,Y 453.517,Z 401.495,A -85,B 0,C 180,E1 -8209.041,E2 -8209.041} C_VEL
LIN {X 0,Y 453.473,Z 401.494,A -85,B 0,C 180,E1 -8211.836,E2 -8211.836} C_VEL
LIN {X 0,Y 453.511,Z 401.496,A -85,B 0,C 180,E1 -8214.734,E2 -8214.734} C_VEL
LIN {X 0,Y 453.534,Z 401.488,A -85,B 0,C 180,E1 -8217.961,E2 -8217.961} C_VEL
LIN {X 0,Y 453.462,Z 401.495,A -85,B 0,C 180,E1 -8221.525,E2 -8221.525} C_VEL
LIN {X 0,Y 453.485,Z 401.496,A -85,B 0,C 180,E1 -8224.778,E2 -8224.778} C_VEL
LIN {X 0,Y 453.476,Z 401.5,A -85,B 0,C 180,E1 -8228.31,E2 -8228.31} C_VEL
LIN {X 0,Y 453.511,Z 401.494,A -85,B 0,C 180,E1 -8230.607,E2 -8230.607} C_VEL
LIN {X 0,Y 453.477,Z 401.493,A -85,B 0,C 180,E1 -8233.248,E2 -8233.248} C_VEL
LIN {X 0,Y 453.461,Z 401.497,A -85,B 0,C 180,E1 -8235.779,E2 -8235.779} C_VEL
LIN {X 0,Y 453.474,Z 401.501,A -85,B 0,C 180,E1 -8238.209,E2 -8238.209} C_VEL
LIN {X 0,Y 453.51,Z 401.491,A -85,B 0,C 180,E1 -8240.79,E2 -8240.79} C_VEL
LIN {X 0,Y 453.452,Z 401.501,A -85,B 0,C 180,E1 -8243.918,E2 -8243.918} C_VEL
LIN {X 0,Y 453.478,Z 401.493,A -85,B 0,C 180,E1 -8247.151,E2 -8247.151} C_VEL
LIN {X 0,Y 453.509,Z 401.495,A -85,B 0,C 180,E1 -8250.271,E2 -8250.271} C_VEL
LIN {X 0,Y 453.504,Z 401.491,A -85,B 0,C 180,E1 -8253.294,E2 -8253.294} C_VEL
LIN {X 0,Y 453.499,Z 401.495,A -85,B 0,C 180,E1 -8256.239,E2 -8256.239} C_VEL
LIN {X 0,Y 453.477,Z 401.494,A -85,B 0,C 180,E1 -8259.118,E2 -8259.118} C_VEL
LIN {X 0,Y 453.508,Z 401.497,A -85,B 0,C 180,E1 -8261.945,E2 -8261.945} C_VEL
LIN {X 0,Y 453.545,Z 401.485,A -85,B 0,C 180,E1 -8264.727,E2 -8264.727} C_VEL
LIN {X 0,Y 453.555,Z 401.485,A -85,B 0,C 180,E1 -8268.379,E2 -8268.379} C_VEL
LIN {X 0,Y 453.648,Z 401.477,A -85,B 0,C 180,E1 -8271.986,E2 -8271.986} C_VEL
LIN {X 0,Y 453.667,Z 401.47,A -85,B 0,C 180,E1 -8274.667,E2 -8274.667} C_VEL
LIN {X 0,Y 453.761,Z 401.462,A -85,B 0,C 180,E1 -8277.337,E2 -8277.337} C_VEL
LIN {X 0,Y 453.82,Z 401.454,A -85,B 0,C 180,E1 -8280,E2 -8280} C_VEL
LIN {X 0,Y 453.762,Z 401.458,A -85,B 0,C 180,E1 -8282.664,E2 -8282.664} C_VEL
LIN {X 0,Y 453.674,Z 401.47,A -85,B 0,C 180,E1 -8286.226,E2 -8286.226} C_VEL
LIN {X 0,Y 453.589,Z 401.481,A -85,B 0,C 180,E1 -8288.914,E2 -8288.914} C_VEL
LIN {X 0,Y 453.56,Z 401.483,A -85,B 0,C 180,E1 -8292.529,E2 -8292.529} C_VEL
LIN {X 0,Y 453.542,Z 401.485,A -85,B 0,C 180,E1 -8296.196,E2 -8296.196} C_VEL
LIN {X 0,Y 453.518,Z 401.493,A -85,B 0,C 180,E1 -8299.041,E2 -8299.041} C_VEL
LIN {X 0,Y 453.474,Z 401.495,A -85,B 0,C 180,E1 -8301.837,E2 -8301.837} C_VEL
LIN {X 0,Y 453.512,Z 401.491,A -85,B 0,C 180,E1 -8304.735,E2 -8304.735} C_VEL
LIN {X 0,Y 453.53,Z 401.487,A -85,B 0,C 180,E1 -8307.96,E2 -8307.96} C_VEL
LIN {X 0,Y 453.465,Z 401.498,A -85,B 0,C 180,E1 -8311.526,E2 -8311.526} C_VEL
LIN {X 0,Y 453.488,Z 401.496,A -85,B 0,C 180,E1 -8314.778,E2 -8314.778} C_VEL
LIN {X 0,Y 453.473,Z 401.499,A -85,B 0,C 180,E1 -8318.311,E2 -8318.311} C_VEL
LIN {X 0,Y 453.494,Z 401.498,A -85,B 0,C 180,E1 -8320.609,E2 -8320.609} C_VEL
LIN {X 0,Y 453.529,Z 401.785,A -85,B 0,C 180,E1 -8321.943,E2 -8321.943} C_VEL
LIN {X 0,Y 454.128,Z 405.669,A -85,B 0,C 180,E1 -8325.389,E2 -8325.389} C_VEL
LIN {X 0,Y 454.491,Z 408.805,A -85,B 0,C 180,E1 -8327.924,E2 -8327.924} C_VEL
LIN {X 0,Y 454.39,Z 412.511,A -85,B 0,C 180,E1 -8330.656,E2 -8330.656} C_VEL
LIN {X 0,Y 454.009,Z 417.347,A -85,B 0,C 180,E1 -8333.969,E2 -8333.969} C_VEL
LIN {X 0,Y 453.697,Z 422.349,A -85,B 0,C 180,E1 -8337.169,E2 -8337.169} C_VEL
LIN {X 0,Y 453.448,Z 427.436,A -85,B 0,C 180,E1 -8340.267,E2 -8340.267} C_VEL
LIN {X 0,Y 453.23,Z 432.624,A -85,B 0,C 180,E1 -8343.277,E2 -8343.277} C_VEL
LIN {X 0,Y 453.027,Z 437.969,A -85,B 0,C 180,E1 -8346.248,E2 -8346.248} C_VEL
LIN {X 0,Y 452.915,Z 443.236,A -85,B 0,C 180,E1 -8349.09,E2 -8349.09} C_VEL
LIN {X 0,Y 452.709,Z 448.61,A -85,B 0,C 180,E1 -8351.912,E2 -8351.912} C_VEL
LIN {X 0,Y 452.665,Z 452.926,A -85,B 0,C 180,E1 -8354.123,E2 -8354.123} C_VEL
LIN {X 0,Y 454.875,Z 464.786,A -85,B 0,C 180,E1 -8354.535,E2 -8354.535} C_VEL
LIN {X 0,Y 456.211,Z 473.709,A -85,B 0,C 180,E1 -8354.932,E2 -8354.932} C_VEL
LIN {X 0,Y 455.996,Z 482.792,A -85,B 0,C 180,E1 -8355.382,E2 -8355.382} C_VEL
LIN {X 0,Y 455.545,Z 491.929,A -85,B 0,C 180,E1 -8355.937,E2 -8355.937} C_VEL
LIN {X 0,Y 455.083,Z 500.93,A -85,B 0,C 180,E1 -8356.606,E2 -8356.606} C_VEL
LIN {X 0,Y 454.743,Z 508.993,A -85,B 0,C 180,E1 -8357.324,E2 -8357.324} C_VEL
LIN {X 0,Y 454.292,Z 517.065,A -85,B 0,C 180,E1 -8358.172,E2 -8358.172} C_VEL
LIN {X 0,Y 453.86,Z 524.287,A -85,B 0,C 180,E1 -8359.065,E2 -8359.065} C_VEL
LIN {X 0,Y 453.536,Z 530.493,A -85,B 0,C 180,E1 -8359.96,E2 -8359.96} C_VEL
LIN {X 0,Y 453.199,Z 537.033,A -85,B 0,C 180,E1 -8361.079,E2 -8361.079} C_VEL
LIN {X 0,Y 452.927,Z 541.535,A -85,B 0,C 180,E1 -8361.972,E2 -8361.972} C_VEL
LIN {X 0,Y 452.724,Z 547.03,A -85,B 0,C 180,E1 -8363.314,E2 -8363.314} C_VEL
LIN {X 0,Y 452.619,Z 551.353,A -85,B 0,C 180,E1 -8364.654,E2 -8364.654} C_VEL
LIN {X 0,Y 452.502,Z 553.717,A -85,B 0,C 180,E1 -8365.546,E2 -8365.546} C_VEL
LIN {X 0,Y 452.489,Z 555.516,A -85,B 0,C 180,E1 -8366.438,E2 -8366.438} C_VEL
LIN {X 0,Y 452.433,Z 557.958,A -85,B 0,C 180,E1 -8368.22,E2 -8368.22} C_VEL
LIN {X 0,Y 452.403,Z 558.545,A -85,B 0,C 180,E1 -8369.11,E2 -8369.11} C_VEL
LIN {X 0,Y 452.403,Z 558.545,A -85,B 0,C 180,E1 -8370.89,E2 -8370.89} C_VEL
LIN {X 0,Y 452.433,Z 557.958,A -85,B 0,C 180,E1 -8371.78,E2 -8371.78} C_VEL
LIN {X 0,Y 452.488,Z 555.516,A -85,B 0,C 180,E1 -8373.562,E2 -8373.562} C_VEL
LIN {X 0,Y 452.567,Z 552.57,A -85,B 0,C 180,E1 -8374.899,E2 -8374.899} C_VEL
LIN {X 0,Y 452.662,Z 548.583,A -85,B 0,C 180,E1 -8376.239,E2 -8376.239} C_VEL
LIN {X 0,Y 452.831,Z 543.452,A -85,B 0,C 180,E1 -8377.58,E2 -8377.58} C_VEL
LIN {X 0,Y 453.114,Z 538.19,A -85,B 0,C 180,E1 -8378.698,E2 -8378.698} C_VEL
LIN {X 0,Y 453.459,Z 531.872,A -85,B 0,C 180,E1 -8379.816,E2 -8379.816} C_VEL
LIN {X 0,Y 453.743,Z 525.917,A -85,B 0,C 180,E1 -8380.711,E2 -8380.711} C_VEL
LIN {X 0,Y 454.143,Z 518.987,A -85,B 0,C 180,E1 -8381.606,E2 -8381.606} C_VEL
LIN {X 0,Y 454.61,Z 510.804,A -85,B 0,C 180,E1 -8382.499,E2 -8382.499} C_VEL
LIN {X 0,Y 455.01,Z 502.609,A -85,B 0,C 180,E1 -8383.255,E2 -8383.255} C_VEL
LIN {X 0,Y 455.488,Z 493.568,A -85,B 0,C 180,E1 -8383.95,E2 -8383.95} C_VEL
LIN {X 0,Y 455.878,Z 484.813,A -85,B 0,C 180,E1 -8384.508,E2 -8384.508} C_VEL
LIN {X 0,Y 456.282,Z 475.01,A -85,B 0,C 180,E1 -8385.008,E2 -8385.008} C_VEL
LIN {X 0,Y 454.907,Z 465.014,A -85,B 0,C 180,E1 -8385.456,E2 -8385.456} C_VEL
LIN {X 0,Y 452.906,Z 454.568,A -85,B 0,C 180,E1 -8385.826,E2 -8385.826} C_VEL
LIN {X 0,Y 452.671,Z 452.934,A -85,B 0,C 180,E1 -8385.872,E2 -8385.872} C_VEL
LIN {X 0,Y 452.776,Z 446.811,A -85,B 0,C 180,E1 -8389.023,E2 -8389.023} C_VEL
LIN {X 0,Y 452.949,Z 441.439,A -85,B 0,C 180,E1 -8391.862,E2 -8391.862} C_VEL
LIN {X 0,Y 453.088,Z 436.119,A -85,B 0,C 180,E1 -8394.759,E2 -8394.759} C_VEL
LIN {X 0,Y 453.32,Z 430.548,A -85,B 0,C 180,E1 -8397.908,E2 -8397.908} C_VEL
LIN {X 0,Y 453.525,Z 425.712,A -85,B 0,C 180,E1 -8400.755,E2 -8400.755} C_VEL
LIN {X 0,Y 453.775,Z 420.643,A -85,B 0,C 180,E1 -8403.887,E2 -8403.887} C_VEL
LIN {X 0,Y 454.127,Z 415.701,A -85,B 0,C 180,E1 -8407.124,E2 -8407.124} C_VEL
LIN {X 0,Y 454.384,Z 412.474,A -85,B 0,C 180,E1 -8409.356,E2 -8409.356} C_VEL
LIN {X 0,Y 454.488,Z 408.806,A -85,B 0,C 180,E1 -8412.076,E2 -8412.076} C_VEL
LIN {X 0,Y 454.13,Z 405.668,A -85,B 0,C 180,E1 -8414.611,E2 -8414.611} C_VEL
LIN {X 0,Y 453.526,Z 401.784,A -85,B 0,C 180,E1 -8418.057,E2 -8418.057} C_VEL
LIN {X 0,Y 453.507,Z 401.497,A -85,B 0,C 180,E1 -8420.79,E2 -8420.79} C_VEL
LIN {X 0,Y 453.454,Z 401.501,A -85,B 0,C 180,E1 -8423.917,E2 -8423.917} C_VEL
LIN {X 0,Y 453.48,Z 401.498,A -85,B 0,C 180,E1 -8427.15,E2 -8427.15} C_VEL
LIN {X 0,Y 453.51,Z 401.491,A -85,B 0,C 180,E1 -8430.27,E2 -8430.27} C_VEL
LIN {X 0,Y 453.505,Z 401.492,A -85,B 0,C 180,E1 -8433.293,E2 -8433.293} C_VEL
LIN {X 0,Y 453.499,Z 401.493,A -85,B 0,C 180,E1 -8436.238,E2 -8436.238} C_VEL
LIN {X 0,Y 453.477,Z 401.496,A -85,B 0,C 180,E1 -8439.117,E2 -8439.117} C_VEL
LIN {X 0,Y 453.506,Z 401.49,A -85,B 0,C 180,E1 -8441.944,E2 -8441.944} C_VEL
LIN {X 0,Y 453.534,Z 401.493,A -85,B 0,C 180,E1 -8444.726,E2 -8444.726} C_VEL
LIN {X 0,Y 453.554,Z 401.489,A -85,B 0,C 180,E1 -8448.378,E2 -8448.378} C_VEL
LIN {X 0,Y 453.646,Z 401.474,A -85,B 0,C 180,E1 -8451.985,E2 -8451.985} C_VEL
LIN {X 0,Y 453.666,Z 401.475,A -85,B 0,C 180,E1 -8454.666,E2 -8454.666} C_VEL
LIN {X 0,Y 453.76,Z 401.458,A -85,B 0,C 180,E1 -8457.336,E2 -8457.336} C_VEL
LIN {X 0,Y 453.817,Z 401.454,A -85,B 0,C 180,E1 -8460,E2 -8460} C_VEL
LIN {X 0,Y 453.759,Z 401.462,A -85,B 0,C 180,E1 -8462.663,E2 -8462.663} C_VEL
LIN {X 0,Y 453.671,Z 401.477,A -85,B 0,C 180,E1 -8466.225,E2 -8466.225} C_VEL
LIN {X 0,Y 453.585,Z 401.481,A -85,B 0,C 180,E1 -8468.913,E2 -8468.913} C_VEL
LIN {X 0,Y 453.556,Z 401.487,A -85,B 0,C 180,E1 -8472.529,E2 -8472.529} C_VEL
LIN {X 0,Y 453.549,Z 401.492,A -85,B 0,C 180,E1 -8476.195,E2 -8476.195} C_VEL
LIN {X 0,Y 453.512,Z 401.489,A -85,B 0,C 180,E1 -8479.04,E2 -8479.04} C_VEL
LIN {X 0,Y 453.469,Z 401.499,A -85,B 0,C 180,E1 -8481.836,E2 -8481.836} C_VEL
LIN {X 0,Y 453.507,Z 401.49,A -85,B 0,C 180,E1 -8484.734,E2 -8484.734} C_VEL
LIN {X 0,Y 453.531,Z 401.495,A -85,B 0,C 180,E1 -8487.961,E2 -8487.961} C_VEL
LIN {X 0,Y 453.476,Z 401.494,A -85,B 0,C 180,E1 -8490.759,E2 -8490.759} C_VEL
LIN {X 0,Y 453.471,Z 401.502,A -85,B 0,C 180,E1 -8493.913,E2 -8493.913} C_VEL
LIN {X 0,Y 453.464,Z 401.496,A -85,B 0,C 180,E1 -8497.188,E2 -8497.188} C_VEL
LIN {X 0,Y 453.526,Z 401.491,A -85,B 0,C 180,E1 -8499.445,E2 -8499.445} C_VEL
LIN {X 0,Y 453.485,Z 401.493,A -85,B 0,C 180,E1 -8502.992,E2 -8502.992} C_VEL
LIN {X 0,Y 453.47,Z 401.501,A -85,B 0,C 180,E1 -8505.781,E2 -8505.781} C_VEL
LIN {X 0,Y 453.49,Z 401.493,A -85,B 0,C 180,E1 -8508.211,E2 -8508.211} C_VEL
LIN {X 0,Y 453.52,Z 401.488,A -85,B 0,C 180,E1 -8510.789,E2 -8510.789} C_VEL
LIN {X 0,Y 453.451,Z 401.5,A -85,B 0,C 180,E1 -8513.918,E2 -8513.918} C_VEL
LIN {X 0,Y 453.477,Z 401.497,A -85,B 0,C 180,E1 -8517.152,E2 -8517.152} C_VEL
LIN {X 0,Y 453.469,Z 401.495,A -85,B 0,C 180,E1 -8520.269,E2 -8520.269} C_VEL
LIN {X 0,Y 453.509,Z 401.496,A -85,B 0,C 180,E1 -8523.295,E2 -8523.295} C_VEL
LIN {X 0,Y 453.498,Z 401.491,A -85,B 0,C 180,E1 -8526.239,E2 -8526.239} C_VEL
LIN {X 0,Y 453.479,Z 401.498,A -85,B 0,C 180,E1 -8529.118,E2 -8529.118} C_VEL
LIN {X 0,Y 453.507,Z 401.494,A -85,B 0,C 180,E1 -8531.945,E2 -8531.945} C_VEL
LIN {X 0,Y 453.536,Z 401.491,A -85,B 0,C 180,E1 -8534.727,E2 -8534.727} C_VEL
LIN {X 0,Y 453.556,Z 401.486,A -85,B 0,C 180,E1 -8538.379,E2 -8538.379} C_VEL
LIN {X 0,Y 453.648,Z 401.476,A -85,B 0,C 180,E1 -8541.985,E2 -8541.985} C_VEL
LIN {X 0,Y 453.633,Z 401.479,A -85,B 0,C 180,E1 -8543.093,E2 -8543.093} C_VEL
LIN {X 0,Y 452.949,Z 401.564,A -85,B 0,C 180,E1 -8543.834,E2 -8543.834} C_VEL
LIN {X 0,Y 450.001,Z 401.935,A -85,B 0,C 180,E1 -8545.035,E2 -8545.035} C_VEL
LIN {X 0,Y 447.577,Z 402.234,A -85,B 0,C 180,E1 -8546.005,E2 -8546.005} C_VEL
LIN {X 0,Y 446.641,Z 402.351,A -85,B 0,C 180,E1 -8546.755,E2 -8546.755} C_VEL
LIN {X 0,Y 446.621,Z 402.353,A -85,B 0,C 180,E1 -8547.008,E2 -8547.008} C_VEL
LIN {X 0,Y 446.791,Z 402.331,A -85,B 0,C 180,E1 -8550,E2 -8550} C_VEL
LIN {X 0,Y 446.706,Z 402.344,A -85,B 0,C 180,E1 -8552.705,E2 -8552.705} C_VEL
LIN {X 0,Y 446.645,Z 402.35,A -85,B 0,C 180,E1 -8556.324,E2 -8556.324} C_VEL
LIN {X 0,Y 446.535,Z 402.364,A -85,B 0,C 180,E1 -8559.055,E2 -8559.055} C_VEL
LIN {X 0,Y 446.518,Z 402.368,A -85,B 0,C 180,E1 -8562.73,E2 -8562.73} C_VEL
LIN {X 0,Y 446.492,Z 402.368,A -85,B 0,C 180,E1 -8566.228,E2 -8566.228} C_VEL
LIN {X 0,Y 446.466,Z 402.37,A -85,B 0,C 180,E1 -8569.303,E2 -8569.303} C_VEL
LIN {X 0,Y 446.415,Z 402.376,A -85,B 0,C 180,E1 -8572.2,E2 -8572.2} C_VEL
LIN {X 0,Y 446.454,Z 402.37,A -85,B 0,C 180,E1 -8575.152,E2 -8575.152} C_VEL
LIN {X 0,Y 446.48,Z 402.368,A -85,B 0,C 180,E1 -8578.179,E2 -8578.179} C_VEL
LIN {X 0,Y 446.416,Z 402.374,A -85,B 0,C 180,E1 -8581.775,E2 -8581.775} C_VEL
LIN {X 0,Y 446.427,Z 402.379,A -85,B 0,C 180,E1 -8584.523,E2 -8584.523} C_VEL
LIN {X 0,Y 446.431,Z 402.375,A -85,B 0,C 180,E1 -8588.083,E2 -8588.083} C_VEL
LIN {X 0,Y 446.442,Z 402.371,A -85,B 0,C 180,E1 -8590.921,E2 -8590.921} C_VEL
LIN {X 0,Y 446.44,Z 402.372,A -85,B 0,C 180,E1 -8593.841,E2 -8593.841} C_VEL
LIN {X 0,Y 446.394,Z 402.382,A -85,B 0,C 180,E1 -8596.403,E2 -8596.403} C_VEL
LIN {X 0,Y 446.422,Z 402.372,A -85,B 0,C 180,E1 -8599.083,E2 -8599.083} C_VEL
LIN {X 0,Y 446.426,Z 402.376,A -85,B 0,C 180,E1 -8601.918,E2 -8601.918} C_VEL
LIN {X 0,Y 446.425,Z 402.373,A -85,B 0,C 180,E1 -8605.477,E2 -8605.477} C_VEL
LIN {X 0,Y 446.426,Z 402.373,A -85,B 0,C 180,E1 -8608.701,E2 -8608.701} C_VEL
LIN {X 0,Y 446.479,Z 402.37,A -85,B 0,C 180,E1 -8611.822,E2 -8611.822} C_VEL
LIN {X 0,Y 446.453,Z 402.369,A -85,B 0,C 180,E1 -8614.848,E2 -8614.848} C_VEL
LIN {X 0,Y 446.443,Z 402.374,A -85,B 0,C 180,E1 -8618.245,E2 -8618.245} C_VEL
LIN {X 0,Y 446.453,Z 402.373,A -85,B 0,C 180,E1 -8621.65,E2 -8621.65} C_VEL
LIN {X 0,Y 446.512,Z 402.362,A -85,B 0,C 180,E1 -8624.48,E2 -8624.48} C_VEL
LIN {X 0,Y 446.513,Z 402.364,A -85,B 0,C 180,E1 -8628.193,E2 -8628.193} C_VEL
LIN {X 0,Y 446.596,Z 402.357,A -85,B 0,C 180,E1 -8631.858,E2 -8631.858} C_VEL
LIN {X 0,Y 446.642,Z 402.345,A -85,B 0,C 180,E1 -8634.583,E2 -8634.583} C_VEL
LIN {X 0,Y 446.705,Z 402.34,A -85,B 0,C 180,E1 -8637.295,E2 -8637.295} C_VEL
LIN {X 0,Y 446.79,Z 402.329,A -85,B 0,C 180,E1 -8640.001,E2 -8640.001} C_VEL
LIN {X 0,Y 446.706,Z 402.337,A -85,B 0,C 180,E1 -8642.706,E2 -8642.706} C_VEL
LIN {X 0,Y 446.643,Z 402.345,A -85,B 0,C 180,E1 -8646.324,E2 -8646.324} C_VEL
LIN {X 0,Y 446.535,Z 402.361,A -85,B 0,C 180,E1 -8649.056,E2 -8649.056} C_VEL
LIN {X 0,Y 446.519,Z 402.361,A -85,B 0,C 180,E1 -8652.73,E2 -8652.73} C_VEL
LIN {X 0,Y 446.494,Z 402.363,A -85,B 0,C 180,E1 -8656.228,E2 -8656.228} C_VEL
LIN {X 0,Y 446.467,Z 402.375,A -85,B 0,C 180,E1 -8659.304,E2 -8659.304} C_VEL
LIN {X 0,Y 446.416,Z 402.373,A -85,B 0,C 180,E1 -8662.2,E2 -8662.2} C_VEL
LIN {X 0,Y 446.456,Z 402.375,A -85,B 0,C 180,E1 -8665.153,E2 -8665.153} C_VEL
LIN {X 0,Y 446.483,Z 402.365,A -85,B 0,C 180,E1 -8668.179,E2 -8668.179} C_VEL
LIN {X 0,Y 446.419,Z 402.374,A -85,B 0,C 180,E1 -8671.776,E2 -8671.776} C_VEL
LIN {X 0,Y 446.429,Z 402.373,A -85,B 0,C 180,E1 -8674.523,E2 -8674.523} C_VEL
LIN {X 0,Y 446.43,Z 402.376,A -85,B 0,C 180,E1 -8678.082,E2 -8678.082} C_VEL
LIN {X 0,Y 446.426,Z 402.38,A -85,B 0,C 180,E1 -8680.918,E2 -8680.918} C_VEL
LIN {X 0,Y 446.434,Z 402.43,A -85,B 0,C 180,E1 -8681.391,E2 -8681.391} C_VEL
LIN {X 0,Y 446.825,Z 405.036,A -85,B 0,C 180,E1 -8683.794,E2 -8683.794} C_VEL
LIN {X 0,Y 447.264,Z 407.917,A -85,B 0,C 180,E1 -8686.288,E2 -8686.288} C_VEL
LIN {X 0,Y 447.489,Z 411.225,A -85,B 0,C 180,E1 -8688.926,E2 -8688.926} C_VEL
LIN {X 0,Y 447.256,Z 415.15,A -85,B 0,C 180,E1 -8691.784,E2 -8691.784} C_VEL
LIN {X 0,Y 446.897,Z 419.691,A -85,B 0,C 180,E1 -8694.862,E2 -8694.862} C_VEL
LIN {X 0,Y 446.609,Z 424.006,A -85,B 0,C 180,E1 -8697.654,E2 -8697.654} C_VEL
LIN {X 0,Y 446.339,Z 429.102,A -85,B 0,C 180,E1 -8700.783,E2 -8700.783} C_VEL
LIN {X 0,Y 446.144,Z 434.388,A -85,B 0,C 180,E1 -8703.885,E2 -8703.885} C_VEL
LIN {X 0,Y 445.91,Z 439.558,A -85,B 0,C 180,E1 -8706.795,E2 -8706.795} C_VEL
